LIN {X 0,Y 150.245,Z 335.769,A -85,B 0,C 180,E1 -24057.283,E2 -24057.283} C_VEL
LIN {X 0,Y 150.219,Z 335.772,A -85,B 0,C 180,E1 -24062.635,E2 -24062.635} C_VEL
LIN {X 0,Y 150.212,Z 335.771,A -85,B 0,C 180,E1 -24067.462,E2 -24067.462} C_VEL
LIN {X 0,Y 150.154,Z 335.78,A -85,B 0,C 180,E1 -24071.507,E2 -24071.507} C_VEL
LIN {X 0,Y 150.127,Z 335.783,A -85,B 0,C 180,E1 -24075.396,E2 -24075.396} C_VEL
LIN {X 0,Y 150.151,Z 335.779,A -85,B 0,C 180,E1 -24079.059,E2 -24079.059} C_VEL
LIN {X 0,Y 150.18,Z 335.776,A -85,B 0,C 180,E1 -24082.708,E2 -24082.708} C_VEL
LIN {X 0,Y 150.217,Z 335.772,A -85,B 0,C 180,E1 -24087.368,E2 -24087.368} C_VEL
LIN {X 0,Y 150.242,Z 335.765,A -85,B 0,C 180,E1 -24092.721,E2 -24092.721} C_VEL
LIN {X 0,Y 150.351,Z 335.756,A -85,B 0,C 180,E1 -24099.21,E2 -24099.21} C_VEL
LIN {X 0,Y 150.349,Z 335.756,A -85,B 0,C 180,E1 -24103.712,E2 -24103.712} C_VEL
LIN {X 0,Y 150.611,Z 335.72,A -85,B 0,C 180,E1 -24109.243,E2 -24109.243} C_VEL
LIN {X 0,Y 150.706,Z 335.711,A -85,B 0,C 180,E1 -24111.958,E2 -24111.958} C_VEL
LIN {X 0,Y 151.217,Z 335.647,A -85,B 0,C 180,E1 -24120,E2 -24120} C_VEL
LIN {X 0,Y 150.703,Z 335.711,A -85,B 0,C 180,E1 -24128.043,E2 -24128.043} C_VEL
LIN {X 0,Y 150.579,Z 335.726,A -85,B 0,C 180,E1 -24131.437,E2 -24131.437} C_VEL
LIN {X 0,Y 150.351,Z 335.755,A -85,B 0,C 180,E1 -24136.288,E2 -24136.288} C_VEL
LIN {X 0,Y 150.351,Z 335.753,A -85,B 0,C 180,E1 -24140.79,E2 -24140.79} C_VEL
LIN {X 0,Y 150.24,Z 335.748,A -85,B 0,C 180,E1 -24147.278,E2 -24147.278} C_VEL
LIN {X 0,Y 150.223,Z 335.774,A -85,B 0,C 180,E1 -24152.636,E2 -24152.636} C_VEL
LIN {X 0,Y 150.407,Z 335.951,A -85,B 0,C 180,E1 -24156.986,E2 -24156.986} C_VEL
LIN {X 0,Y 151.096,Z 339.515,A -85,B 0,C 180,E1 -24161.908,E2 -24161.908} C_VEL
LIN {X 0,Y 151.984,Z 343.974,A -85,B 0,C 180,E1 -24167.721,E2 -24167.721} C_VEL
LIN {X 0,Y 152.438,Z 347.108,A -85,B 0,C 180,E1 -24171.608,E2 -24171.608} C_VEL
LIN {X 0,Y 152.098,Z 348.347,A -85,B 0,C 180,E1 -24173.08,E2 -24173.08} C_VEL
LIN {X 0,Y 153.587,Z 362.688,A -85,B 0,C 180,E1 -24174.817,E2 -24174.817} C_VEL
LIN {X 0,Y 154.517,Z 375.98,A -85,B 0,C 180,E1 -24176.92,E2 -24176.92} C_VEL
LIN {X 0,Y 154.934,Z 388.273,A -85,B 0,C 180,E1 -24179.322,E2 -24179.322} C_VEL
LIN {X 0,Y 155.055,Z 399.237,A -85,B 0,C 180,E1 -24181.949,E2 -24181.949} C_VEL
LIN {X 0,Y 154.986,Z 410.057,A -85,B 0,C 180,E1 -24185.085,E2 -24185.085} C_VEL
LIN {X 0,Y 152.696,Z 419.643,A -85,B 0,C 180,E1 -24188.395,E2 -24188.395} C_VEL
LIN {X 0,Y 150.671,Z 428.608,A -85,B 0,C 180,E1 -24192.351,E2 -24192.351} C_VEL
LIN {X 0,Y 149.307,Z 435.832,A -85,B 0,C 180,E1 -24196.387,E2 -24196.387} C_VEL
LIN {X 0,Y 148.638,Z 441.612,A -85,B 0,C 180,E1 -24200.474,E2 -24200.474} C_VEL
LIN {X 0,Y 148.521,Z 446.113,A -85,B 0,C 180,E1 -24204.569,E2 -24204.569} C_VEL
LIN {X 0,Y 148.533,Z 448.434,A -85,B 0,C 180,E1 -24207.288,E2 -24207.288} C_VEL
LIN {X 0,Y 148.892,Z 450.302,A -85,B 0,C 180,E1 -24210,E2 -24210} C_VEL
LIN {X 0,Y 148.189,Z 452.535,A -85,B 0,C 180,E1 -24215.443,E2 -24215.443} C_VEL
LIN {X 0,Y 148.386,Z 453.179,A -85,B 0,C 180,E1 -24220.921,E2 -24220.921} C_VEL
LIN {X 0,Y 149.84,Z 452.386,A -85,B 0,C 180,E1 -24226.345,E2 -24226.345} C_VEL
LIN {X 0,Y 152.88,Z 450.2,A -85,B 0,C 180,E1 -24231.578,E2 -24231.578} C_VEL
LIN {X 0,Y 157.193,Z 446.504,A -85,B 0,C 180,E1 -24236.558,E2 -24236.558} C_VEL
LIN {X 0,Y 162.714,Z 441.245,A -85,B 0,C 180,E1 -24241.219,E2 -24241.219} C_VEL
LIN {X 0,Y 167.836,Z 436.146,A -85,B 0,C 180,E1 -24244.424,E2 -24244.424} C_VEL
LIN {X 0,Y 173.282,Z 429.984,A -85,B 0,C 180,E1 -24247.472,E2 -24247.472} C_VEL
LIN {X 0,Y 177.395,Z 423.553,A -85,B 0,C 180,E1 -24250.386,E2 -24250.386} C_VEL
LIN {X 0,Y 181.085,Z 416.172,A -85,B 0,C 180,E1 -24253.543,E2 -24253.543} C_VEL
LIN {X 0,Y 184.291,Z 407.788,A -85,B 0,C 180,E1 -24257.04,E2 -24257.04} C_VEL
LIN {X 0,Y 185.114,Z 404.915,A -85,B 0,C 180,E1 -24258.355,E2 -24258.355} C_VEL
LIN {X 0,Y 185.083,Z 402.347,A -85,B 0,C 180,E1 -24260.006,E2 -24260.006} C_VEL
LIN {X 0,Y 184.494,Z 400.473,A -85,B 0,C 180,E1 -24261.729,E2 -24261.729} C_VEL
LIN {X 0,Y 183.298,Z 399.467,A -85,B 0,C 180,E1 -24263.517,E2 -24263.517} C_VEL
LIN {X 0,Y 180.117,Z 398.092,A -85,B 0,C 180,E1 -24268.479,E2 -24268.479} C_VEL
LIN {X 0,Y 179.921,Z 397.396,A -85,B 0,C 180,E1 -24269.74,E2 -24269.74} C_VEL
LIN {X 0,Y 180.125,Z 395.776,A -85,B 0,C 180,E1 -24272.082,E2 -24272.082} C_VEL
LIN {X 0,Y 180.229,Z 394.714,A -85,B 0,C 180,E1 -24274.599,E2 -24274.599} C_VEL
LIN {X 0,Y 180.436,Z 394.168,A -85,B 0,C 180,E1 -24277.076,E2 -24277.076} C_VEL
LIN {X 0,Y 180.637,Z 394.859,A -85,B 0,C 180,E1 -24281.865,E2 -24281.865} C_VEL
LIN {X 0,Y 180.986,Z 395.569,A -85,B 0,C 180,E1 -24284.227,E2 -24284.227} C_VEL
LIN {X 0,Y 181.604,Z 398.314,A -85,B 0,C 180,E1 -24288.843,E2 -24288.843} C_VEL
LIN {X 0,Y 181.83,Z 401.361,A -85,B 0,C 180,E1 -24292.225,E2 -24292.225} C_VEL
LIN {X 0,Y 181.689,Z 403.801,A -85,B 0,C 180,E1 -24294.45,E2 -24294.45} C_VEL
LIN {X 0,Y 180.97,Z 407.418,A -85,B 0,C 180,E1 -24297.217,E2 -24297.217} C_VEL
LIN {X 0,Y 174.553,Z 414.57,A -85,B 0,C 180,E1 -24300,E2 -24300} C_VEL
LIN {X 0,Y 168.875,Z 420.089,A -85,B 0,C 180,E1 -24302.801,E2 -24302.801} C_VEL
LIN {X 0,Y 162.669,Z 425.365,A -85,B 0,C 180,E1 -24306.432,E2 -24306.432} C_VEL
LIN {X 0,Y 157.159,Z 429.256,A -85,B 0,C 180,E1 -24310.319,E2 -24310.319} C_VEL
LIN {X 0,Y 152.408,Z 431.935,A -85,B 0,C 180,E1 -24314.446,E2 -24314.446} C_VEL
LIN {X 0,Y 148.044,Z 433.624,A -85,B 0,C 180,E1 -24319.409,E2 -24319.409} C_VEL
LIN {X 0,Y 145.416,Z 433.971,A -85,B 0,C 180,E1 -24323.324,E2 -24323.324} C_VEL
LIN {X 0,Y 143.173,Z 433.396,A -85,B 0,C 180,E1 -24327.923,E2 -24327.923} C_VEL
LIN {X 0,Y 141.605,Z 431.564,A -85,B 0,C 180,E1 -24333.089,E2 -24333.089} C_VEL
LIN {X 0,Y 140.981,Z 428.174,A -85,B 0,C 180,E1 -24338.658,E2 -24338.658} C_VEL
LIN {X 0,Y 141.387,Z 423.269,A -85,B 0,C 180,E1 -24344.099,E2 -24344.099} C_VEL
LIN {X 0,Y 142.458,Z 417.277,A -85,B 0,C 180,E1 -24349.049,E2 -24349.049} C_VEL
LIN {X 0,Y 143.968,Z 410.137,A -85,B 0,C 180,E1 -24353.584,E2 -24353.584} C_VEL
LIN {X 0,Y 145.907,Z 402.46,A -85,B 0,C 180,E1 -24357.46,E2 -24357.46} C_VEL
LIN {X 0,Y 148.171,Z 393.253,A -85,B 0,C 180,E1 -24361.187,E2 -24361.187} C_VEL
LIN {X 0,Y 150.589,Z 383.793,A -85,B 0,C 180,E1 -24364.237,E2 -24364.237} C_VEL
LIN {X 0,Y 153.429,Z 371.561,A -85,B 0,C 180,E1 -24367.335,E2 -24367.335} C_VEL
LIN {X 0,Y 152.432,Z 365.897,A -85,B 0,C 180,E1 -24368.821,E2 -24368.821} C_VEL
LIN {X 0,Y 149.531,Z 354.899,A -85,B 0,C 180,E1 -24371.503,E2 -24371.503} C_VEL
LIN {X 0,Y 146.011,Z 344.016,A -85,B 0,C 180,E1 -24373.86,E2 -24373.86} C_VEL
LIN {X 0,Y 143.361,Z 336.628,A -85,B 0,C 180,E1 -24375.358,E2 -24375.358} C_VEL
LIN {X 0,Y 143.529,Z 336.608,A -85,B 0,C 180,E1 -24378.705,E2 -24378.705} C_VEL
LIN {X 0,Y 143.622,Z 336.6,A -85,B 0,C 180,E1 -24381.558,E2 -24381.558} C_VEL
LIN {X 0,Y 144.176,Z 336.519,A -85,B 0,C 180,E1 -24390,E2 -24390} C_VEL
LIN {X 0,Y 143.623,Z 336.592,A -85,B 0,C 180,E1 -24398.442,E2 -24398.442} C_VEL
LIN {X 0,Y 143.505,Z 336.609,A -85,B 0,C 180,E1 -24401.63,E2 -24401.63} C_VEL
LIN {X 0,Y 143.302,Z 336.634,A -85,B 0,C 180,E1 -24407.113,E2 -24407.113} C_VEL
LIN {X 0,Y 143.277,Z 336.633,A -85,B 0,C 180,E1 -24411.255,E2 -24411.255} C_VEL
LIN {X 0,Y 143.191,Z 336.649,A -85,B 0,C 180,E1 -24417.938,E2 -24417.938} C_VEL
LIN {X 0,Y 143.17,Z 336.65,A -85,B 0,C 180,E1 -24423.436,E2 -24423.436} C_VEL
LIN {X 0,Y 143.076,Z 336.658,A -85,B 0,C 180,E1 -24429.686,E2 -24429.686} C_VEL
LIN {X 0,Y 143.057,Z 336.665,A -85,B 0,C 180,E1 -24433.455,E2 -24433.455} C_VEL
LIN {X 0,Y 143.066,Z 336.658,A -85,B 0,C 180,E1 -24437.465,E2 -24437.465} C_VEL
LIN {X 0,Y 143.078,Z 336.662,A -85,B 0,C 180,E1 -24441.806,E2 -24441.806} C_VEL
LIN {X 0,Y 143.184,Z 336.648,A -85,B 0,C 180,E1 -24447.322,E2 -24447.322} C_VEL
LIN {X 0,Y 143.19,Z 336.644,A -85,B 0,C 180,E1 -24452.065,E2 -24452.065} C_VEL
LIN {X 0,Y 143.276,Z 336.637,A -85,B 0,C 180,E1 -24458.748,E2 -24458.748} C_VEL
LIN {X 0,Y 143.293,Z 336.632,A -85,B 0,C 180,E1 -24462.886,E2 -24462.886} C_VEL
LIN {X 0,Y 143.537,Z 336.602,A -85,B 0,C 180,E1 -24468.706,E2 -24468.706} C_VEL
LIN {X 0,Y 143.627,Z 336.593,A -85,B 0,C 180,E1 -24471.559,E2 -24471.559} C_VEL
LIN {X 0,Y 144.176,Z 336.524,A -85,B 0,C 180,E1 -24480,E2 -24480} C_VEL
LIN {X 0,Y 143.625,Z 336.593,A -85,B 0,C 180,E1 -24488.442,E2 -24488.442} C_VEL
LIN {X 0,Y 143.506,Z 336.607,A -85,B 0,C 180,E1 -24491.628,E2 -24491.628} C_VEL
LIN {X 0,Y 143.294,Z 336.635,A -85,B 0,C 180,E1 -24497.114,E2 -24497.114} C_VEL
LIN {X 0,Y 143.276,Z 336.633,A -85,B 0,C 180,E1 -24501.252,E2 -24501.252} C_VEL
LIN {X 0,Y 143.185,Z 336.629,A -85,B 0,C 180,E1 -24507.931,E2 -24507.931} C_VEL
LIN {X 0,Y 143.166,Z 336.653,A -85,B 0,C 180,E1 -24513.432,E2 -24513.432} C_VEL
LIN {X 0,Y 143.365,Z 336.834,A -85,B 0,C 180,E1 -24516.853,E2 -24516.853} C_VEL
LIN {X 0,Y 144.161,Z 341.144,A -85,B 0,C 180,E1 -24523.041,E2 -24523.041} C_VEL
LIN {X 0,Y 145.132,Z 345.655,A -85,B 0,C 180,E1 -24529.112,E2 -24529.112} C_VEL
LIN {X 0,Y 145.245,Z 347.987,A -85,B 0,C 180,E1 -24531.942,E2 -24531.942} C_VEL
LIN {X 0,Y 146.713,Z 360.951,A -85,B 0,C 180,E1 -24533.592,E2 -24533.592} C_VEL
LIN {X 0,Y 147.528,Z 374.304,A -85,B 0,C 180,E1 -24535.755,E2 -24535.755} C_VEL
LIN {X 0,Y 147.979,Z 385.945,A -85,B 0,C 180,E1 -24538.105,E2 -24538.105} C_VEL
LIN {X 0,Y 148.086,Z 397.385,A -85,B 0,C 180,E1 -24540.892,E2 -24540.892} C_VEL
LIN {X 0,Y 147.962,Z 408.129,A -85,B 0,C 180,E1 -24544.08,E2 -24544.08} C_VEL
LIN {X 0,Y 147.523,Z 411.986,A -85,B 0,C 180,E1 -24545.364,E2 -24545.364} C_VEL
LIN {X 0,Y 145.267,Z 420.792,A -85,B 0,C 180,E1 -24548.725,E2 -24548.725} C_VEL
LIN {X 0,Y 143.333,Z 429.463,A -85,B 0,C 180,E1 -24552.891,E2 -24552.891} C_VEL
LIN {X 0,Y 142.059,Z 436.408,A -85,B 0,C 180,E1 -24557.137,E2 -24557.137} C_VEL
LIN {X 0,Y 141.52,Z 441.927,A -85,B 0,C 180,E1 -24561.432,E2 -24561.432} C_VEL
LIN {X 0,Y 141.463,Z 446.196,A -85,B 0,C 180,E1 -24565.726,E2 -24565.726} C_VEL
LIN {X 0,Y 141.835,Z 449.329,A -85,B 0,C 180,E1 -24570,E2 -24570} C_VEL
LIN {X 0,Y 141.128,Z 451.694,A -85,B 0,C 180,E1 -24575.716,E2 -24575.716} C_VEL
LIN {X 0,Y 141.379,Z 452.562,A -85,B 0,C 180,E1 -24581.469,E2 -24581.469} C_VEL
LIN {X 0,Y 143.005,Z 451.956,A -85,B 0,C 180,E1 -24587.15,E2 -24587.15} C_VEL
LIN {X 0,Y 146.274,Z 449.958,A -85,B 0,C 180,E1 -24592.605,E2 -24592.605} C_VEL
LIN {X 0,Y 150.864,Z 446.527,A -85,B 0,C 180,E1 -24597.765,E2 -24597.765} C_VEL
LIN {X 0,Y 156.7,Z 441.521,A -85,B 0,C 180,E1 -24602.562,E2 -24602.562} C_VEL
LIN {X 0,Y 162.052,Z 436.665,A -85,B 0,C 180,E1 -24605.837,E2 -24605.837} C_VEL
LIN {X 0,Y 166.846,Z 431.825,A -85,B 0,C 180,E1 -24608.412,E2 -24608.412} C_VEL
LIN {X 0,Y 170.928,Z 426.317,A -85,B 0,C 180,E1 -24611.138,E2 -24611.138} C_VEL
LIN {X 0,Y 174.605,Z 420.247,A -85,B 0,C 180,E1 -24613.974,E2 -24613.974} C_VEL
LIN {X 0,Y 178.166,Z 412.97,A -85,B 0,C 180,E1 -24617.252,E2 -24617.252} C_VEL
LIN {X 0,Y 179.764,Z 408.96,A -85,B 0,C 180,E1 -24619.128,E2 -24619.128} C_VEL
LIN {X 0,Y 179.932,Z 405.737,A -85,B 0,C 180,E1 -24621.37,E2 -24621.37} C_VEL
LIN {X 0,Y 180.007,Z 401.346,A -85,B 0,C 180,E1 -24625.076,E2 -24625.076} C_VEL
LIN {X 0,Y 179.942,Z 399.637,A -85,B 0,C 180,E1 -24626.852,E2 -24626.852} C_VEL
LIN {X 0,Y 179.921,Z 397.396,A -85,B 0,C 180,E1 -24629.74,E2 -24629.74} C_VEL
LIN {X 0,Y 179.547,Z 396.738,A -85,B 0,C 180,E1 -24631.606,E2 -24631.606} C_VEL
LIN {X 0,Y 178.617,Z 397.022,A -85,B 0,C 180,E1 -24633.485,E2 -24633.485} C_VEL
LIN {X 0,Y 175.965,Z 399.453,A -85,B 0,C 180,E1 -24638.586,E2 -24638.586} C_VEL
LIN {X 0,Y 175.774,Z 399.815,A -85,B 0,C 180,E1 -24639.901,E2 -24639.901} C_VEL
LIN {X 0,Y 176.108,Z 400.68,A -85,B 0,C 180,E1 -24643.778,E2 -24643.778} C_VEL
LIN {X 0,Y 176.294,Z 401.749,A -85,B 0,C 180,E1 -24646.161,E2 -24646.161} C_VEL
LIN {X 0,Y 176.472,Z 403.124,A -85,B 0,C 180,E1 -24648.514,E2 -24648.514} C_VEL
LIN {X 0,Y 176.408,Z 405.939,A -85,B 0,C 180,E1 -24651.984,E2 -24651.984} C_VEL
LIN {X 0,Y 175.999,Z 408.249,A -85,B 0,C 180,E1 -24654.27,E2 -24654.27} C_VEL
LIN {X 0,Y 175.402,Z 410.284,A -85,B 0,C 180,E1 -24655.979,E2 -24655.979} C_VEL
LIN {X 0,Y 167.712,Z 417.965,A -85,B 0,C 180,E1 -24659.253,E2 -24659.253} C_VEL
LIN {X 0,Y 161.208,Z 423.488,A -85,B 0,C 180,E1 -24662.498,E2 -24662.498} C_VEL
LIN {X 0,Y 155.456,Z 427.697,A -85,B 0,C 180,E1 -24665.953,E2 -24665.953} C_VEL
LIN {X 0,Y 149.863,Z 431.104,A -85,B 0,C 180,E1 -24669.992,E2 -24669.992} C_VEL
LIN {X 0,Y 145.055,Z 433.318,A -85,B 0,C 180,E1 -24674.299,E2 -24674.299} C_VEL
LIN {X 0,Y 141.099,Z 434.435,A -85,B 0,C 180,E1 -24678.848,E2 -24678.848} C_VEL
LIN {X 0,Y 137.749,Z 434.434,A -85,B 0,C 180,E1 -24684.089,E2 -24684.089} C_VEL
LIN {X 0,Y 135.809,Z 433.538,A -85,B 0,C 180,E1 -24688.389,E2 -24688.389} C_VEL
LIN {X 0,Y 134.464,Z 431.572,A -85,B 0,C 180,E1 -24693.251,E2 -24693.251} C_VEL
LIN {X 0,Y 133.878,Z 427.9,A -85,B 0,C 180,E1 -24699.046,E2 -24699.046} C_VEL
LIN {X 0,Y 134.418,Z 422.569,A -85,B 0,C 180,E1 -24704.897,E2 -24704.897} C_VEL
LIN {X 0,Y 135.591,Z 416.362,A -85,B 0,C 180,E1 -24709.941,E2 -24709.941} C_VEL
LIN {X 0,Y 137.354,Z 408.436,A -85,B 0,C 180,E1 -24714.951,E2 -24714.951} C_VEL
LIN {X 0,Y 139.457,Z 400.349,A -85,B 0,C 180,E1 -24718.95,E2 -24718.95} C_VEL
LIN {X 0,Y 142.096,Z 390.282,A -85,B 0,C 180,E1 -24722.907,E2 -24722.907} C_VEL
LIN {X 0,Y 144.743,Z 379.879,A -85,B 0,C 180,E1 -24726.136,E2 -24726.136} C_VEL
LIN {X 0,Y 146.341,Z 373.192,A -85,B 0,C 180,E1 -24727.835,E2 -24727.835} C_VEL
LIN {X 0,Y 146.462,Z 371.459,A -85,B 0,C 180,E1 -24728.281,E2 -24728.281} C_VEL
LIN {X 0,Y 144.025,Z 360.858,A -85,B 0,C 180,E1 -24731.138,E2 -24731.138} C_VEL
LIN {X 0,Y 140.443,Z 348.913,A -85,B 0,C 180,E1 -24734.024,E2 -24734.024} C_VEL
LIN {X 0,Y 136.353,Z 337.528,A -85,B 0,C 180,E1 -24736.531,E2 -24736.531} C_VEL
LIN {X 0,Y 136.547,Z 337.483,A -85,B 0,C 180,E1 -24741.117,E2 -24741.117} C_VEL
LIN {X 0,Y 137.133,Z 337.396,A -85,B 0,C 180,E1 -24750,E2 -24750} C_VEL
LIN {X 0,Y 136.55,Z 337.475,A -85,B 0,C 180,E1 -24758.882,E2 -24758.882} C_VEL
LIN {X 0,Y 136.441,Z 337.489,A -85,B 0,C 180,E1 -24761.89,E2 -24761.89} C_VEL
LIN {X 0,Y 136.243,Z 337.514,A -85,B 0,C 180,E1 -24768.03,E2 -24768.03} C_VEL
LIN {X 0,Y 136.199,Z 337.515,A -85,B 0,C 180,E1 -24771.749,E2 -24771.749} C_VEL
LIN {X 0,Y 136.101,Z 337.529,A -85,B 0,C 180,E1 -24778.617,E2 -24778.617} C_VEL
LIN {X 0,Y 136.079,Z 337.534,A -85,B 0,C 180,E1 -24784.619,E2 -24784.619} C_VEL
LIN {X 0,Y 136.051,Z 337.532,A -85,B 0,C 180,E1 -24789.208,E2 -24789.208} C_VEL
LIN {X 0,Y 135.999,Z 337.545,A -85,B 0,C 180,E1 -24793.658,E2 -24793.658} C_VEL
LIN {X 0,Y 136.005,Z 337.539,A -85,B 0,C 180,E1 -24797.797,E2 -24797.797} C_VEL
LIN {X 0,Y 136.028,Z 337.541,A -85,B 0,C 180,E1 -24801.685,E2 -24801.685} C_VEL
LIN {X 0,Y 136.056,Z 337.533,A -85,B 0,C 180,E1 -24805.74,E2 -24805.74} C_VEL
LIN {X 0,Y 136.145,Z 337.521,A -85,B 0,C 180,E1 -24812.317,E2 -24812.317} C_VEL
LIN {X 0,Y 136.243,Z 337.513,A -85,B 0,C 180,E1 -24818.833,E2 -24818.833} C_VEL
LIN {X 0,Y 136.246,Z 337.514,A -85,B 0,C 180,E1 -24825.054,E2 -24825.054} C_VEL
LIN {X 0,Y 136.427,Z 337.487,A -85,B 0,C 180,E1 -24828.178,E2 -24828.178} C_VEL
LIN {X 0,Y 136.552,Z 337.473,A -85,B 0,C 180,E1 -24831.118,E2 -24831.118} C_VEL
LIN {X 0,Y 137.133,Z 337.401,A -85,B 0,C 180,E1 -24840,E2 -24840} C_VEL
LIN {X 0,Y 136.551,Z 337.476,A -85,B 0,C 180,E1 -24848.883,E2 -24848.883} C_VEL
LIN {X 0,Y 136.442,Z 337.487,A -85,B 0,C 180,E1 -24851.891,E2 -24851.891} C_VEL
LIN {X 0,Y 136.238,Z 337.514,A -85,B 0,C 180,E1 -24858.031,E2 -24858.031} C_VEL
LIN {X 0,Y 136.197,Z 337.515,A -85,B 0,C 180,E1 -24861.746,E2 -24861.746} C_VEL
LIN {X 0,Y 136.094,Z 337.515,A -85,B 0,C 180,E1 -24868.61,E2 -24868.61} C_VEL
LIN {X 0,Y 136.322,Z 337.618,A -85,B 0,C 180,E1 -24876.591,E2 -24876.591} C_VEL
LIN {X 0,Y 136.947,Z 341.085,A -85,B 0,C 180,E1 -24881.848,E2 -24881.848} C_VEL
LIN {X 0,Y 137.946,Z 345.763,A -85,B 0,C 180,E1 -24888.523,E2 -24888.523} C_VEL
LIN {X 0,Y 138.196,Z 347.298,A -85,B 0,C 180,E1 -24890.634,E2 -24890.634} C_VEL
LIN {X 0,Y 139.643,Z 357.54,A -85,B 0,C 180,E1 -24892.052,E2 -24892.052} C_VEL
LIN {X 0,Y 140.584,Z 370.636,A -85,B 0,C 180,E1 -24894.158,E2 -24894.158} C_VEL
LIN {X 0,Y 141.026,Z 381.698,A -85,B 0,C 180,E1 -24896.351,E2 -24896.351} C_VEL
LIN {X 0,Y 141.176,Z 393.28,A -85,B 0,C 180,E1 -24899.14,E2 -24899.14} C_VEL
LIN {X 0,Y 141.021,Z 404.853,A -85,B 0,C 180,E1 -24902.549,E2 -24902.549} C_VEL
LIN {X 0,Y 140.782,Z 410.704,A -85,B 0,C 180,E1 -24904.544,E2 -24904.544} C_VEL
LIN {X 0,Y 138.239,Z 420.331,A -85,B 0,C 180,E1 -24908.371,E2 -24908.371} C_VEL
LIN {X 0,Y 136.262,Z 428.973,A -85,B 0,C 180,E1 -24912.748,E2 -24912.748} C_VEL
LIN {X 0,Y 134.996,Z 435.881,A -85,B 0,C 180,E1 -24917.217,E2 -24917.217} C_VEL
LIN {X 0,Y 134.465,Z 442.154,A -85,B 0,C 180,E1 -24922.493,E2 -24922.493} C_VEL
LIN {X 0,Y 134.455,Z 446.187,A -85,B 0,C 180,E1 -24927.004,E2 -24927.004} C_VEL
LIN {X 0,Y 134.78,Z 448.284,A -85,B 0,C 180,E1 -24930,E2 -24930} C_VEL
LIN {X 0,Y 134.122,Z 450.673,A -85,B 0,C 180,E1 -24935.369,E2 -24935.369} C_VEL
LIN {X 0,Y 134.097,Z 451.549,A -85,B 0,C 180,E1 -24939.046,E2 -24939.046} C_VEL
LIN {X 0,Y 135.12,Z 451.865,A -85,B 0,C 180,E1 -24945.074,E2 -24945.074} C_VEL
LIN {X 0,Y 137.813,Z 450.799,A -85,B 0,C 180,E1 -24950.915,E2 -24950.915} C_VEL
LIN {X 0,Y 142.041,Z 448.286,A -85,B 0,C 180,E1 -24956.443,E2 -24956.443} C_VEL
LIN {X 0,Y 147.522,Z 444.355,A -85,B 0,C 180,E1 -24961.604,E2 -24961.604} C_VEL
LIN {X 0,Y 152.538,Z 440.353,A -85,B 0,C 180,E1 -24965.165,E2 -24965.165} C_VEL
LIN {X 0,Y 158.383,Z 435.381,A -85,B 0,C 180,E1 -24968.406,E2 -24968.406} C_VEL
LIN {X 0,Y 162.259,Z 431.556,A -85,B 0,C 180,E1 -24970.52,E2 -24970.52} C_VEL
LIN {X 0,Y 166.675,Z 425.883,A -85,B 0,C 180,E1 -24973.488,E2 -24973.488} C_VEL
LIN {X 0,Y 170.991,Z 419.074,A -85,B 0,C 180,E1 -24976.85,E2 -24976.85} C_VEL
LIN {X 0,Y 174.308,Z 412.689,A -85,B 0,C 180,E1 -24980.003,E2 -24980.003} C_VEL
LIN {X 0,Y 174.842,Z 408.305,A -85,B 0,C 180,E1 -24983.507,E2 -24983.507} C_VEL
LIN {X 0,Y 174.992,Z 405.928,A -85,B 0,C 180,E1 -24985.787,E2 -24985.787} C_VEL
LIN {X 0,Y 175.135,Z 402.528,A -85,B 0,C 180,E1 -24990.17,E2 -24990.17} C_VEL
LIN {X 0,Y 175.375,Z 401.39,A -85,B 0,C 180,E1 -24991.841,E2 -24991.841} C_VEL
LIN {X 0,Y 175.572,Z 400.417,A -85,B 0,C 180,E1 -24993.875,E2 -24993.875} C_VEL
LIN {X 0,Y 175.793,Z 399.63,A -85,B 0,C 180,E1 -24996.856,E2 -24996.856} C_VEL
LIN {X 0,Y 175.774,Z 399.815,A -85,B 0,C 180,E1 -24999.901,E2 -24999.901} C_VEL
LIN {X 0,Y 175.394,Z 400.701,A -85,B 0,C 180,E1 -25001.803,E2 -25001.803} C_VEL
LIN {X 0,Y 174.352,Z 402.414,A -85,B 0,C 180,E1 -25003.643,E2 -25003.643} C_VEL
LIN {X 0,Y 171.237,Z 407.858,A -85,B 0,C 180,E1 -25008.563,E2 -25008.563} C_VEL
LIN {X 0,Y 170.97,Z 408.845,A -85,B 0,C 180,E1 -25009.863,E2 -25009.863} C_VEL
LIN {X 0,Y 170.559,Z 411.305,A -85,B 0,C 180,E1 -25012.899,E2 -25012.899} C_VEL
LIN {X 0,Y 170.12,Z 412.478,A -85,B 0,C 180,E1 -25014.073,E2 -25014.073} C_VEL
LIN {X 0,Y 169.36,Z 413.599,A -85,B 0,C 180,E1 -25014.839,E2 -25014.839} C_VEL
LIN {X 0,Y 161.74,Z 420.404,A -85,B 0,C 180,E1 -25018.04,E2 -25018.04} C_VEL
LIN {X 0,Y 154.674,Z 425.775,A -85,B 0,C 180,E1 -25021.547,E2 -25021.547} C_VEL
LIN {X 0,Y 148.23,Z 429.87,A -85,B 0,C 180,E1 -25025.441,E2 -25025.441} C_VEL
LIN {X 0,Y 142.563,Z 432.736,A -85,B 0,C 180,E1 -25029.613,E2 -25029.613} C_VEL
LIN {X 0,Y 136.998,Z 434.685,A -85,B 0,C 180,E1 -25034.862,E2 -25034.862} C_VEL
LIN {X 0,Y 133.7,Z 435.214,A -85,B 0,C 180,E1 -25038.882,E2 -25038.882} C_VEL
LIN {X 0,Y 130.63,Z 434.873,A -85,B 0,C 180,E1 -25043.848,E2 -25043.848} C_VEL
LIN {X 0,Y 128.24,Z 433.274,A -85,B 0,C 180,E1 -25049.553,E2 -25049.553} C_VEL
LIN {X 0,Y 126.993,Z 430.189,A -85,B 0,C 180,E1 -25055.672,E2 -25055.672} C_VEL
LIN {X 0,Y 126.91,Z 425.77,A -85,B 0,C 180,E1 -25061.646,E2 -25061.646} C_VEL
LIN {X 0,Y 127.755,Z 419.993,A -85,B 0,C 180,E1 -25067.318,E2 -25067.318} C_VEL
LIN {X 0,Y 128.951,Z 414.346,A -85,B 0,C 180,E1 -25071.669,E2 -25071.669} C_VEL
LIN {X 0,Y 131.038,Z 405.803,A -85,B 0,C 180,E1 -25076.86,E2 -25076.86} C_VEL
LIN {X 0,Y 133.206,Z 397.599,A -85,B 0,C 180,E1 -25080.788,E2 -25080.788} C_VEL
LIN {X 0,Y 136.129,Z 386.982,A -85,B 0,C 180,E1 -25084.79,E2 -25084.79} C_VEL
LIN {X 0,Y 139.023,Z 375.735,A -85,B 0,C 180,E1 -25088.11,E2 -25088.11} C_VEL
LIN {X 0,Y 139.524,Z 372.436,A -85,B 0,C 180,E1 -25088.967,E2 -25088.967} C_VEL
LIN {X 0,Y 137.02,Z 361.66,A -85,B 0,C 180,E1 -25092.076,E2 -25092.076} C_VEL
LIN {X 0,Y 133.465,Z 349.866,A -85,B 0,C 180,E1 -25095.145,E2 -25095.145} C_VEL
LIN {X 0,Y 129.463,Z 338.909,A -85,B 0,C 180,E1 -25097.726,E2 -25097.726} C_VEL
LIN {X 0,Y 129.369,Z 338.373,A -85,B 0,C 180,E1 -25097.917,E2 -25097.917} C_VEL
LIN {X 0,Y 129.47,Z 338.363,A -85,B 0,C 180,E1 -25100.628,E2 -25100.628} C_VEL
LIN {X 0,Y 130.088,Z 338.273,A -85,B 0,C 180,E1 -25110,E2 -25110} C_VEL
LIN {X 0,Y 129.473,Z 338.356,A -85,B 0,C 180,E1 -25119.372,E2 -25119.372} C_VEL
LIN {X 0,Y 129.344,Z 338.372,A -85,B 0,C 180,E1 -25122.553,E2 -25122.553} C_VEL
LIN {X 0,Y 129.154,Z 338.396,A -85,B 0,C 180,E1 -25129.056,E2 -25129.056} C_VEL
LIN {X 0,Y 129.109,Z 338.397,A -85,B 0,C 180,E1 -25132.398,E2 -25132.398} C_VEL
LIN {X 0,Y 129.036,Z 338.408,A -85,B 0,C 180,E1 -25139.374,E2 -25139.374} C_VEL
LIN {X 0,Y 128.993,Z 338.416,A -85,B 0,C 180,E1 -25145.19,E2 -25145.19} C_VEL
LIN {X 0,Y 128.951,Z 338.42,A -85,B 0,C 180,E1 -25150.845,E2 -25150.845} C_VEL
LIN {X 0,Y 128.922,Z 338.424,A -85,B 0,C 180,E1 -25155.128,E2 -25155.128} C_VEL
LIN {X 0,Y 128.943,Z 338.423,A -85,B 0,C 180,E1 -25159.736,E2 -25159.736} C_VEL
LIN {X 0,Y 128.96,Z 338.415,A -85,B 0,C 180,E1 -25164.832,E2 -25164.832} C_VEL
LIN {X 0,Y 129.017,Z 338.413,A -85,B 0,C 180,E1 -25170.643,E2 -25170.643} C_VEL
LIN {X 0,Y 129.028,Z 338.409,A -85,B 0,C 180,E1 -25174.167,E2 -25174.167} C_VEL
LIN {X 0,Y 129.108,Z 338.402,A -85,B 0,C 180,E1 -25177.729,E2 -25177.729} C_VEL
LIN {X 0,Y 129.149,Z 338.392,A -85,B 0,C 180,E1 -25180.944,E2 -25180.944} C_VEL
LIN {X 0,Y 129.35,Z 338.369,A -85,B 0,C 180,E1 -25187.962,E2 -25187.962} C_VEL
LIN {X 0,Y 129.474,Z 338.353,A -85,B 0,C 180,E1 -25190.628,E2 -25190.628} C_VEL
LIN {X 0,Y 130.088,Z 338.279,A -85,B 0,C 180,E1 -25200,E2 -25200} C_VEL
LIN {X 0,Y 129.474,Z 338.357,A -85,B 0,C 180,E1 -25209.372,E2 -25209.372} C_VEL
LIN {X 0,Y 129.345,Z 338.37,A -85,B 0,C 180,E1 -25212.553,E2 -25212.553} C_VEL
LIN {X 0,Y 129.15,Z 338.396,A -85,B 0,C 180,E1 -25219.057,E2 -25219.057} C_VEL
LIN {X 0,Y 129.109,Z 338.393,A -85,B 0,C 180,E1 -25222.399,E2 -25222.399} C_VEL
LIN {X 0,Y 129.018,Z 338.401,A -85,B 0,C 180,E1 -25229.358,E2 -25229.358} C_VEL
LIN {X 0,Y 129.26,Z 338.501,A -85,B 0,C 180,E1 -25236.512,E2 -25236.512} C_VEL
LIN {X 0,Y 129.963,Z 342.288,A -85,B 0,C 180,E1 -25242.527,E2 -25242.527} C_VEL
LIN {X 0,Y 130.933,Z 346.6,A -85,B 0,C 180,E1 -25248.988,E2 -25248.988} C_VEL
LIN {X 0,Y 130.954,Z 346.811,A -85,B 0,C 180,E1 -25249.227,E2 -25249.227} C_VEL
LIN {X 0,Y 132.554,Z 353.665,A -85,B 0,C 180,E1 -25250.31,E2 -25250.31} C_VEL
LIN {X 0,Y 133.597,Z 366.413,A -85,B 0,C 180,E1 -25252.354,E2 -25252.354} C_VEL
LIN {X 0,Y 134.128,Z 380.26,A -85,B 0,C 180,E1 -25255.155,E2 -25255.155} C_VEL
LIN {X 0,Y 134.213,Z 391.447,A -85,B 0,C 180,E1 -25257.928,E2 -25257.928} C_VEL
LIN {X 0,Y 134.018,Z 402.963,A -85,B 0,C 180,E1 -25261.411,E2 -25261.411} C_VEL
LIN {X 0,Y 133.82,Z 410.05,A -85,B 0,C 180,E1 -25263.925,E2 -25263.925} C_VEL
LIN {X 0,Y 131.671,Z 418.151,A -85,B 0,C 180,E1 -25267.234,E2 -25267.234} C_VEL
LIN {X 0,Y 129.483,Z 427.047,A -85,B 0,C 180,E1 -25271.814,E2 -25271.814} C_VEL
LIN {X 0,Y 128.095,Z 434.223,A -85,B 0,C 180,E1 -25276.516,E2 -25276.516} C_VEL
LIN {X 0,Y 127.509,Z 439.074,A -85,B 0,C 180,E1 -25280.482,E2 -25280.482} C_VEL
LIN {X 0,Y 127.423,Z 443.727,A -85,B 0,C 180,E1 -25285.254,E2 -25285.254} C_VEL
LIN {X 0,Y 127.727,Z 447.194,A -85,B 0,C 180,E1 -25290,E2 -25290} C_VEL
LIN {X 0,Y 127.09,Z 449.685,A -85,B 0,C 180,E1 -25295.501,E2 -25295.501} C_VEL
LIN {X 0,Y 127.067,Z 450.769,A -85,B 0,C 180,E1 -25299.551,E2 -25299.551} C_VEL
LIN {X 0,Y 128.263,Z 451.265,A -85,B 0,C 180,E1 -25305.901,E2 -25305.901} C_VEL
LIN {X 0,Y 131.188,Z 450.4,A -85,B 0,C 180,E1 -25312.025,E2 -25312.025} C_VEL
LIN {X 0,Y 135.68,Z 448.166,A -85,B 0,C 180,E1 -25317.787,E2 -25317.787} C_VEL
LIN {X 0,Y 141.511,Z 444.442,A -85,B 0,C 180,E1 -25323.114,E2 -25323.114} C_VEL
LIN {X 0,Y 146.809,Z 440.693,A -85,B 0,C 180,E1 -25326.756,E2 -25326.756} C_VEL
LIN {X 0,Y 155.016,Z 434.187,A -85,B 0,C 180,E1 -25331.102,E2 -25331.102} C_VEL
LIN {X 0,Y 159.595,Z 429.313,A -85,B 0,C 180,E1 -25333.914,E2 -25333.914} C_VEL
LIN {X 0,Y 164.613,Z 422.835,A -85,B 0,C 180,E1 -25337.432,E2 -25337.432} C_VEL
LIN {X 0,Y 168.221,Z 417.117,A -85,B 0,C 180,E1 -25340.433,E2 -25340.433} C_VEL
LIN {X 0,Y 168.896,Z 415.672,A -85,B 0,C 180,E1 -25341.378,E2 -25341.378} C_VEL
LIN {X 0,Y 169.519,Z 412.195,A -85,B 0,C 180,E1 -25344.52,E2 -25344.52} C_VEL
LIN {X 0,Y 169.9,Z 409.553,A -85,B 0,C 180,E1 -25347.469,E2 -25347.469} C_VEL
LIN {X 0,Y 170.515,Z 405.984,A -85,B 0,C 180,E1 -25353.039,E2 -25353.039} C_VEL
LIN {X 0,Y 170.739,Z 405.044,A -85,B 0,C 180,E1 -25355.693,E2 -25355.693} C_VEL
LIN {X 0,Y 170.857,Z 404.775,A -85,B 0,C 180,E1 -25358.271,E2 -25358.271} C_VEL
LIN {X 0,Y 171.015,Z 405.55,A -85,B 0,C 180,E1 -25363.281,E2 -25363.281} C_VEL
LIN {X 0,Y 171.061,Z 406.44,A -85,B 0,C 180,E1 -25365.729,E2 -25365.729} C_VEL
LIN {X 0,Y 171.135,Z 407.696,A -85,B 0,C 180,E1 -25368.151,E2 -25368.151} C_VEL
LIN {X 0,Y 170.97,Z 408.845,A -85,B 0,C 180,E1 -25369.863,E2 -25369.863} C_VEL
LIN {X 0,Y 170.417,Z 409.969,A -85,B 0,C 180,E1 -25370.867,E2 -25370.867} C_VEL
LIN {X 0,Y 168.478,Z 412.255,A -85,B 0,C 180,E1 -25372.055,E2 -25372.055} C_VEL
LIN {X 0,Y 163.485,Z 416.775,A -85,B 0,C 180,E1 -25373.751,E2 -25373.751} C_VEL
LIN {X 0,Y 159.984,Z 419.601,A -85,B 0,C 180,E1 -25374.972,E2 -25374.972} C_VEL
LIN {X 0,Y 151.698,Z 425.682,A -85,B 0,C 180,E1 -25378.672,E2 -25378.672} C_VEL
LIN {X 0,Y 144.199,Z 430.216,A -85,B 0,C 180,E1 -25382.793,E2 -25382.793} C_VEL
LIN {X 0,Y 139.683,Z 432.476,A -85,B 0,C 180,E1 -25385.775,E2 -25385.775} C_VEL
LIN {X 0,Y 135.264,Z 434.212,A -85,B 0,C 180,E1 -25389.174,E2 -25389.174} C_VEL
LIN {X 0,Y 130.319,Z 435.525,A -85,B 0,C 180,E1 -25393.895,E2 -25393.895} C_VEL
LIN {X 0,Y 125.808,Z 435.787,A -85,B 0,C 180,E1 -25399.583,E2 -25399.583} C_VEL
LIN {X 0,Y 123.216,Z 435.061,A -85,B 0,C 180,E1 -25404.13,E2 -25404.13} C_VEL
LIN {X 0,Y 121.109,Z 433.322,A -85,B 0,C 180,E1 -25409.488,E2 -25409.488} C_VEL
LIN {X 0,Y 119.869,Z 430.002,A -85,B 0,C 180,E1 -25415.895,E2 -25415.895} C_VEL
LIN {X 0,Y 119.866,Z 425.056,A -85,B 0,C 180,E1 -25422.395,E2 -25422.395} C_VEL
LIN {X 0,Y 120.805,Z 419.293,A -85,B 0,C 180,E1 -25428.067,E2 -25428.067} C_VEL
LIN {X 0,Y 122.381,Z 412.128,A -85,B 0,C 180,E1 -25433.511,E2 -25433.511} C_VEL
LIN {X 0,Y 124.826,Z 403.093,A -85,B 0,C 180,E1 -25438.826,E2 -25438.826} C_VEL
LIN {X 0,Y 127.411,Z 393.625,A -85,B 0,C 180,E1 -25443.176,E2 -25443.176} C_VEL
LIN {X 0,Y 130.312,Z 383.378,A -85,B 0,C 180,E1 -25446.844,E2 -25446.844} C_VEL
LIN {X 0,Y 132.668,Z 374.294,A -85,B 0,C 180,E1 -25449.454,E2 -25449.454} C_VEL
LIN {X 0,Y 130.837,Z 365.442,A -85,B 0,C 180,E1 -25452.207,E2 -25452.207} C_VEL
LIN {X 0,Y 127.371,Z 353.38,A -85,B 0,C 180,E1 -25455.623,E2 -25455.623} C_VEL
LIN {X 0,Y 122.964,Z 341.423,A -85,B 0,C 180,E1 -25458.773,E2 -25458.773} C_VEL
LIN {X 0,Y 122.352,Z 339.247,A -85,B 0,C 180,E1 -25459.284,E2 -25459.284} C_VEL
LIN {X 0,Y 122.595,Z 339.217,A -85,B 0,C 180,E1 -25466.714,E2 -25466.714} C_VEL
LIN {X 0,Y 123.041,Z 339.15,A -85,B 0,C 180,E1 -25470,E2 -25470} C_VEL
LIN {X 0,Y 122.422,Z 339.234,A -85,B 0,C 180,E1 -25476.593,E2 -25476.593} C_VEL
LIN {X 0,Y 122.409,Z 339.237,A -85,B 0,C 180,E1 -25479.918,E2 -25479.918} C_VEL
LIN {X 0,Y 122.24,Z 339.255,A -85,B 0,C 180,E1 -25483.296,E2 -25483.296} C_VEL
LIN {X 0,Y 122.046,Z 339.281,A -85,B 0,C 180,E1 -25490.213,E2 -25490.213} C_VEL
LIN {X 0,Y 121.984,Z 339.286,A -85,B 0,C 180,E1 -25493.785,E2 -25493.785} C_VEL
LIN {X 0,Y 121.942,Z 339.29,A -85,B 0,C 180,E1 -25500.174,E2 -25500.174} C_VEL
LIN {X 0,Y 121.913,Z 339.297,A -85,B 0,C 180,E1 -25506.19,E2 -25506.19} C_VEL
LIN {X 0,Y 121.885,Z 339.301,A -85,B 0,C 180,E1 -25511.445,E2 -25511.445} C_VEL
LIN {X 0,Y 121.873,Z 339.302,A -85,B 0,C 180,E1 -25518.562,E2 -25518.562} C_VEL
LIN {X 0,Y 121.912,Z 339.293,A -85,B 0,C 180,E1 -25524.797,E2 -25524.797} C_VEL
LIN {X 0,Y 121.927,Z 339.297,A -85,B 0,C 180,E1 -25529.839,E2 -25529.839} C_VEL
LIN {X 0,Y 121.983,Z 339.289,A -85,B 0,C 180,E1 -25536.216,E2 -25536.216} C_VEL
LIN {X 0,Y 122.043,Z 339.279,A -85,B 0,C 180,E1 -25539.787,E2 -25539.787} C_VEL
LIN {X 0,Y 122.098,Z 339.274,A -85,B 0,C 180,E1 -25543.274,E2 -25543.274} C_VEL
LIN {X 0,Y 122.401,Z 339.233,A -85,B 0,C 180,E1 -25550.082,E2 -25550.082} C_VEL
LIN {X 0,Y 122.599,Z 339.209,A -85,B 0,C 180,E1 -25556.714,E2 -25556.714} C_VEL
LIN {X 0,Y 123.041,Z 339.157,A -85,B 0,C 180,E1 -25560,E2 -25560} C_VEL
LIN {X 0,Y 122.419,Z 339.23,A -85,B 0,C 180,E1 -25566.594,E2 -25566.594} C_VEL
LIN {X 0,Y 122.324,Z 339.245,A -85,B 0,C 180,E1 -25572.386,E2 -25572.386} C_VEL
LIN {X 0,Y 122.105,Z 339.275,A -85,B 0,C 180,E1 -25576.726,E2 -25576.726} C_VEL
LIN {X 0,Y 122.028,Z 339.273,A -85,B 0,C 180,E1 -25582.854,E2 -25582.854} C_VEL
LIN {X 0,Y 121.936,Z 339.287,A -85,B 0,C 180,E1 -25590.167,E2 -25590.167} C_VEL
LIN {X 0,Y 122.222,Z 339.332,A -85,B 0,C 180,E1 -25596.386,E2 -25596.386} C_VEL
LIN {X 0,Y 122.982,Z 343.481,A -85,B 0,C 180,E1 -25603.296,E2 -25603.296} C_VEL
LIN {X 0,Y 123.632,Z 346.293,A -85,B 0,C 180,E1 -25607.647,E2 -25607.647} C_VEL
LIN {X 0,Y 124.595,Z 349.556,A -85,B 0,C 180,E1 -25608.214,E2 -25608.214} C_VEL
LIN {X 0,Y 126.087,Z 355.337,A -85,B 0,C 180,E1 -25609.263,E2 -25609.263} C_VEL
LIN {X 0,Y 126.931,Z 367.414,A -85,B 0,C 180,E1 -25611.379,E2 -25611.379} C_VEL
LIN {X 0,Y 127.294,Z 380.275,A -85,B 0,C 180,E1 -25614.167,E2 -25614.167} C_VEL
LIN {X 0,Y 127.304,Z 392.466,A -85,B 0,C 180,E1 -25617.434,E2 -25617.434} C_VEL
LIN {X 0,Y 127.024,Z 402.995,A -85,B 0,C 180,E1 -25620.854,E2 -25620.854} C_VEL
LIN {X 0,Y 126.686,Z 410.363,A -85,B 0,C 180,E1 -25623.653,E2 -25623.653} C_VEL
LIN {X 0,Y 124.232,Z 419.134,A -85,B 0,C 180,E1 -25627.551,E2 -25627.551} C_VEL
LIN {X 0,Y 122.154,Z 427.771,A -85,B 0,C 180,E1 -25632.419,E2 -25632.419} C_VEL
LIN {X 0,Y 120.848,Z 434.692,A -85,B 0,C 180,E1 -25637.403,E2 -25637.403} C_VEL
LIN {X 0,Y 120.386,Z 440.64,A -85,B 0,C 180,E1 -25642.954,E2 -25642.954} C_VEL
LIN {X 0,Y 120.505,Z 444.965,A -85,B 0,C 180,E1 -25648.329,E2 -25648.329} C_VEL
LIN {X 0,Y 120.677,Z 446.073,A -85,B 0,C 180,E1 -25650,E2 -25650} C_VEL
LIN {X 0,Y 120.063,Z 448.678,A -85,B 0,C 180,E1 -25655.664,E2 -25655.664} C_VEL
LIN {X 0,Y 120.059,Z 449.919,A -85,B 0,C 180,E1 -25660.114,E2 -25660.114} C_VEL
LIN {X 0,Y 121.421,Z 450.658,A -85,B 0,C 180,E1 -25666.823,E2 -25666.823} C_VEL
LIN {X 0,Y 124.621,Z 449.992,A -85,B 0,C 180,E1 -25673.252,E2 -25673.252} C_VEL
LIN {X 0,Y 129.407,Z 447.96,A -85,B 0,C 180,E1 -25679.261,E2 -25679.261} C_VEL
LIN {X 0,Y 135.597,Z 444.566,A -85,B 0,C 180,E1 -25684.76,E2 -25684.76} C_VEL
LIN {X 0,Y 141.194,Z 441.003,A -85,B 0,C 180,E1 -25688.477,E2 -25688.477} C_VEL
LIN {X 0,Y 147.565,Z 436.511,A -85,B 0,C 180,E1 -25691.819,E2 -25691.819} C_VEL
LIN {X 0,Y 151.746,Z 433.063,A -85,B 0,C 180,E1 -25694.005,E2 -25694.005} C_VEL
LIN {X 0,Y 157.424,Z 427.017,A -85,B 0,C 180,E1 -25697.658,E2 -25697.658} C_VEL
LIN {X 0,Y 162.269,Z 420.769,A -85,B 0,C 180,E1 -25701.224,E2 -25701.224} C_VEL
LIN {X 0,Y 163.047,Z 419.572,A -85,B 0,C 180,E1 -25701.986,E2 -25701.986} C_VEL
LIN {X 0,Y 163.858,Z 416.822,A -85,B 0,C 180,E1 -25704.58,E2 -25704.58} C_VEL
LIN {X 0,Y 164.213,Z 415.357,A -85,B 0,C 180,E1 -25706.194,E2 -25706.194} C_VEL
LIN {X 0,Y 164.634,Z 413.184,A -85,B 0,C 180,E1 -25709.185,E2 -25709.185} C_VEL
LIN {X 0,Y 165.304,Z 410.829,A -85,B 0,C 180,E1 -25713.232,E2 -25713.232} C_VEL
LIN {X 0,Y 165.496,Z 410.192,A -85,B 0,C 180,E1 -25714.87,E2 -25714.87} C_VEL
LIN {X 0,Y 165.656,Z 409.686,A -85,B 0,C 180,E1 -25718.965,E2 -25718.965} C_VEL
LIN {X 0,Y 165.689,Z 410.174,A -85,B 0,C 180,E1 -25722.727,E2 -25722.727} C_VEL
LIN {X 0,Y 165.648,Z 410.903,A -85,B 0,C 180,E1 -25725.252,E2 -25725.252} C_VEL
LIN {X 0,Y 165.613,Z 412.016,A -85,B 0,C 180,E1 -25727.749,E2 -25727.749} C_VEL
LIN {X 0,Y 165.28,Z 413.457,A -85,B 0,C 180,E1 -25730.207,E2 -25730.207} C_VEL
LIN {X 0,Y 164.624,Z 415.328,A -85,B 0,C 180,E1 -25732.641,E2 -25732.641} C_VEL
LIN {X 0,Y 164.186,Z 416.036,A -85,B 0,C 180,E1 -25733.33,E2 -25733.33} C_VEL
LIN {X 0,Y 159.984,Z 419.601,A -85,B 0,C 180,E1 -25734.972,E2 -25734.972} C_VEL
LIN {X 0,Y 156.135,Z 422.407,A -85,B 0,C 180,E1 -25736.258,E2 -25736.258} C_VEL
LIN {X 0,Y 148.621,Z 426.782,A -85,B 0,C 180,E1 -25738.06,E2 -25738.06} C_VEL
LIN {X 0,Y 141.114,Z 430.449,A -85,B 0,C 180,E1 -25740.138,E2 -25740.138} C_VEL
LIN {X 0,Y 137.372,Z 432.11,A -85,B 0,C 180,E1 -25741.867,E2 -25741.867} C_VEL
LIN {X 0,Y 131.076,Z 434.597,A -85,B 0,C 180,E1 -25746.156,E2 -25746.156} C_VEL
LIN {X 0,Y 126.981,Z 435.768,A -85,B 0,C 180,E1 -25749.557,E2 -25749.557} C_VEL
LIN {X 0,Y 122.934,Z 436.391,A -85,B 0,C 180,E1 -25753.619,E2 -25753.619} C_VEL
LIN {X 0,Y 118.859,Z 436.248,A -85,B 0,C 180,E1 -25758.902,E2 -25758.902} C_VEL
LIN {X 0,Y 115.466,Z 434.874,A -85,B 0,C 180,E1 -25765.218,E2 -25765.218} C_VEL
LIN {X 0,Y 113.356,Z 432.097,A -85,B 0,C 180,E1 -25771.951,E2 -25771.951} C_VEL
LIN {X 0,Y 112.602,Z 427.977,A -85,B 0,C 180,E1 -25778.619,E2 -25778.619} C_VEL
LIN {X 0,Y 113.101,Z 422.506,A -85,B 0,C 180,E1 -25785.141,E2 -25785.141} C_VEL
LIN {X 0,Y 114.476,Z 415.795,A -85,B 0,C 180,E1 -25791.158,E2 -25791.158} C_VEL
LIN {X 0,Y 116.186,Z 408.876,A -85,B 0,C 180,E1 -25796.049,E2 -25796.049} C_VEL
LIN {X 0,Y 118.551,Z 400.606,A -85,B 0,C 180,E1 -25800.72,E2 -25800.72} C_VEL
LIN {X 0,Y 121.437,Z 390.61,A -85,B 0,C 180,E1 -25805.191,E2 -25805.191} C_VEL
LIN {X 0,Y 124.469,Z 379.873,A -85,B 0,C 180,E1 -25808.902,E2 -25808.902} C_VEL
LIN {X 0,Y 125.753,Z 374.703,A -85,B 0,C 180,E1 -25810.408,E2 -25810.408} C_VEL
LIN {X 0,Y 123.615,Z 365.409,A -85,B 0,C 180,E1 -25813.485,E2 -25813.485} C_VEL
LIN {X 0,Y 120.762,Z 355.428,A -85,B 0,C 180,E1 -25816.539,E2 -25816.539} C_VEL
LIN {X 0,Y 116.492,Z 343.375,A -85,B 0,C 180,E1 -25820.011,E2 -25820.011} C_VEL
LIN {X 0,Y 115.35,Z 340.124,A -85,B 0,C 180,E1 -25820.907,E2 -25820.907} C_VEL
LIN {X 0,Y 115.993,Z 340.028,A -85,B 0,C 180,E1 -25830,E2 -25830} C_VEL
LIN {X 0,Y 115.363,Z 340.112,A -85,B 0,C 180,E1 -25836.998,E2 -25836.998} C_VEL
LIN {X 0,Y 115.249,Z 340.127,A -85,B 0,C 180,E1 -25842.66,E2 -25842.66} C_VEL
LIN {X 0,Y 115.012,Z 340.158,A -85,B 0,C 180,E1 -25847.79,E2 -25847.79} C_VEL
LIN {X 0,Y 114.947,Z 340.162,A -85,B 0,C 180,E1 -25853.493,E2 -25853.493} C_VEL
LIN {X 0,Y 114.869,Z 340.171,A -85,B 0,C 180,E1 -25861.069,E2 -25861.069} C_VEL
LIN {X 0,Y 114.803,Z 340.18,A -85,B 0,C 180,E1 -25867.748,E2 -25867.748} C_VEL
LIN {X 0,Y 114.795,Z 340.185,A -85,B 0,C 180,E1 -25872.722,E2 -25872.722} C_VEL
LIN {X 0,Y 114.795,Z 340.18,A -85,B 0,C 180,E1 -25877.667,E2 -25877.667} C_VEL
LIN {X 0,Y 114.789,Z 340.185,A -85,B 0,C 180,E1 -25882.744,E2 -25882.744} C_VEL
LIN {X 0,Y 114.857,Z 340.178,A -85,B 0,C 180,E1 -25888.943,E2 -25888.943} C_VEL
LIN {X 0,Y 114.948,Z 340.166,A -85,B 0,C 180,E1 -25896.508,E2 -25896.508} C_VEL
LIN {X 0,Y 115.005,Z 340.155,A -85,B 0,C 180,E1 -25902.209,E2 -25902.209} C_VEL
LIN {X 0,Y 115.313,Z 340.115,A -85,B 0,C 180,E1 -25909.465,E2 -25909.465} C_VEL
LIN {X 0,Y 115.523,Z 340.091,A -85,B 0,C 180,E1 -25916.513,E2 -25916.513} C_VEL
LIN {X 0,Y 115.992,Z 340.035,A -85,B 0,C 180,E1 -25920,E2 -25920} C_VEL
LIN {X 0,Y 115.361,Z 340.111,A -85,B 0,C 180,E1 -25926.999,E2 -25926.999} C_VEL
LIN {X 0,Y 115.257,Z 340.123,A -85,B 0,C 180,E1 -25932.673,E2 -25932.673} C_VEL
LIN {X 0,Y 115.009,Z 340.158,A -85,B 0,C 180,E1 -25937.791,E2 -25937.791} C_VEL
LIN {X 0,Y 114.946,Z 340.151,A -85,B 0,C 180,E1 -25943.489,E2 -25943.489} C_VEL
LIN {X 0,Y 114.878,Z 340.171,A -85,B 0,C 180,E1 -25951.074,E2 -25951.074} C_VEL
LIN {X 0,Y 115.183,Z 340.285,A -85,B 0,C 180,E1 -25956.506,E2 -25956.506} C_VEL
LIN {X 0,Y 115.911,Z 344.155,A -85,B 0,C 180,E1 -25963.315,E2 -25963.315} C_VEL
LIN {X 0,Y 116.26,Z 345.614,A -85,B 0,C 180,E1 -25965.803,E2 -25965.803} C_VEL
LIN {X 0,Y 117.374,Z 349.206,A -85,B 0,C 180,E1 -25966.551,E2 -25966.551} C_VEL
LIN {X 0,Y 119.587,Z 356.882,A -85,B 0,C 180,E1 -25968.163,E2 -25968.163} C_VEL
LIN {X 0,Y 120.282,Z 369.27,A -85,B 0,C 180,E1 -25970.549,E2 -25970.549} C_VEL
LIN {X 0,Y 120.488,Z 380.919,A -85,B 0,C 180,E1 -25973.282,E2 -25973.282} C_VEL
LIN {X 0,Y 120.364,Z 393.142,A -85,B 0,C 180,E1 -25976.811,E2 -25976.811} C_VEL
LIN {X 0,Y 119.988,Z 403.881,A -85,B 0,C 180,E1 -25980.565,E2 -25980.565} C_VEL
LIN {X 0,Y 119.719,Z 409.709,A -85,B 0,C 180,E1 -25982.938,E2 -25982.938} C_VEL
LIN {X 0,Y 117.26,Z 418.488,A -85,B 0,C 180,E1 -25987.072,E2 -25987.072} C_VEL
LIN {X 0,Y 115.106,Z 427.101,A -85,B 0,C 180,E1 -25992.225,E2 -25992.225} C_VEL
LIN {X 0,Y 113.789,Z 434.017,A -85,B 0,C 180,E1 -25997.516,E2 -25997.516} C_VEL
LIN {X 0,Y 113.364,Z 439.508,A -85,B 0,C 180,E1 -26002.878,E2 -26002.878} C_VEL
LIN {X 0,Y 113.471,Z 443.731,A -85,B 0,C 180,E1 -26008.225,E2 -26008.225} C_VEL
LIN {X 0,Y 113.647,Z 444.876,A -85,B 0,C 180,E1 -26010,E2 -26010} C_VEL
LIN {X 0,Y 113.045,Z 447.625,A -85,B 0,C 180,E1 -26015.887,E2 -26015.887} C_VEL
LIN {X 0,Y 113.077,Z 449.039,A -85,B 0,C 180,E1 -26020.746,E2 -26020.746} C_VEL
LIN {X 0,Y 114.622,Z 449.966,A -85,B 0,C 180,E1 -26027.853,E2 -26027.853} C_VEL
LIN {X 0,Y 118.104,Z 449.564,A -85,B 0,C 180,E1 -26034.617,E2 -26034.617} C_VEL
LIN {X 0,Y 123.231,Z 447.774,A -85,B 0,C 180,E1 -26040.883,E2 -26040.883} C_VEL
LIN {X 0,Y 129.821,Z 444.601,A -85,B 0,C 180,E1 -26046.548,E2 -26046.548} C_VEL
LIN {X 0,Y 137.874,Z 439.996,A -85,B 0,C 180,E1 -26051.504,E2 -26051.504} C_VEL
LIN {X 0,Y 144.628,Z 435.47,A -85,B 0,C 180,E1 -26054.798,E2 -26054.798} C_VEL
LIN {X 0,Y 148.659,Z 432.044,A -85,B 0,C 180,E1 -26057.12,E2 -26057.12} C_VEL
LIN {X 0,Y 154.297,Z 426.316,A -85,B 0,C 180,E1 -26060.744,E2 -26060.744} C_VEL
LIN {X 0,Y 156.054,Z 424.298,A -85,B 0,C 180,E1 -26062.011,E2 -26062.011} C_VEL
LIN {X 0,Y 157.536,Z 422.304,A -85,B 0,C 180,E1 -26063.42,E2 -26063.42} C_VEL
LIN {X 0,Y 158.437,Z 419.713,A -85,B 0,C 180,E1 -26066.326,E2 -26066.326} C_VEL
LIN {X 0,Y 159.287,Z 416.689,A -85,B 0,C 180,E1 -26070.965,E2 -26070.965} C_VEL
LIN {X 0,Y 159.946,Z 415.178,A -85,B 0,C 180,E1 -26073.934,E2 -26073.934} C_VEL
LIN {X 0,Y 160.183,Z 414.411,A -85,B 0,C 180,E1 -26077.128,E2 -26077.128} C_VEL
LIN {X 0,Y 160.217,Z 414.302,A -85,B 0,C 180,E1 -26079.456,E2 -26079.456} C_VEL
LIN {X 0,Y 160.139,Z 414.561,A -85,B 0,C 180,E1 -26082.109,E2 -26082.109} C_VEL
LIN {X 0,Y 160.052,Z 415.234,A -85,B 0,C 180,E1 -26085.026,E2 -26085.026} C_VEL
LIN {X 0,Y 159.921,Z 416.064,A -85,B 0,C 180,E1 -26087.306,E2 -26087.306} C_VEL
LIN {X 0,Y 159.424,Z 417.396,A -85,B 0,C 180,E1 -26089.843,E2 -26089.843} C_VEL
LIN {X 0,Y 158.994,Z 418.239,A -85,B 0,C 180,E1 -26091.1,E2 -26091.1} C_VEL
LIN {X 0,Y 157.517,Z 419.677,A -85,B 0,C 180,E1 -26092.307,E2 -26092.307} C_VEL
LIN {X 0,Y 149.701,Z 425.28,A -85,B 0,C 180,E1 -26095.462,E2 -26095.462} C_VEL
LIN {X 0,Y 143.128,Z 429.217,A -85,B 0,C 180,E1 -26098.585,E2 -26098.585} C_VEL
LIN {X 0,Y 137.372,Z 432.11,A -85,B 0,C 180,E1 -26101.867,E2 -26101.867} C_VEL
LIN {X 0,Y 133.704,Z 433.561,A -85,B 0,C 180,E1 -26103.738,E2 -26103.738} C_VEL
LIN {X 0,Y 126.488,Z 435.588,A -85,B 0,C 180,E1 -26106.608,E2 -26106.608} C_VEL
LIN {X 0,Y 119.557,Z 436.834,A -85,B 0,C 180,E1 -26109.85,E2 -26109.85} C_VEL
LIN {X 0,Y 116.452,Z 437.047,A -85,B 0,C 180,E1 -26112.28,E2 -26112.28} C_VEL
LIN {X 0,Y 111.433,Z 436.528,A -85,B 0,C 180,E1 -26118.906,E2 -26118.906} C_VEL
LIN {X 0,Y 108.397,Z 434.975,A -85,B 0,C 180,E1 -26124.809,E2 -26124.809} C_VEL
LIN {X 0,Y 106.22,Z 431.884,A -85,B 0,C 180,E1 -26131.959,E2 -26131.959} C_VEL
LIN {X 0,Y 105.526,Z 427.347,A -85,B 0,C 180,E1 -26139.247,E2 -26139.247} C_VEL
LIN {X 0,Y 105.937,Z 422.863,A -85,B 0,C 180,E1 -26144.708,E2 -26144.708} C_VEL
LIN {X 0,Y 107.025,Z 417.319,A -85,B 0,C 180,E1 -26150.12,E2 -26150.12} C_VEL
LIN {X 0,Y 108.959,Z 409.608,A -85,B 0,C 180,E1 -26156.067,E2 -26156.067} C_VEL
LIN {X 0,Y 111.741,Z 400.142,A -85,B 0,C 180,E1 -26161.706,E2 -26161.706} C_VEL
LIN {X 0,Y 114.442,Z 391.112,A -85,B 0,C 180,E1 -26165.914,E2 -26165.914} C_VEL
LIN {X 0,Y 117.283,Z 381.592,A -85,B 0,C 180,E1 -26169.426,E2 -26169.426} C_VEL
LIN {X 0,Y 118.825,Z 376.031,A -85,B 0,C 180,E1 -26171.143,E2 -26171.143} C_VEL
LIN {X 0,Y 116.815,Z 366.776,A -85,B 0,C 180,E1 -26174.445,E2 -26174.445} C_VEL
LIN {X 0,Y 114.169,Z 357.444,A -85,B 0,C 180,E1 -26177.558,E2 -26177.558} C_VEL
LIN {X 0,Y 110.528,Z 346.836,A -85,B 0,C 180,E1 -26180.853,E2 -26180.853} C_VEL
LIN {X 0,Y 108.301,Z 340.995,A -85,B 0,C 180,E1 -26182.66,E2 -26182.66} C_VEL
LIN {X 0,Y 108.918,Z 340.909,A -85,B 0,C 180,E1 -26190,E2 -26190} C_VEL
LIN {X 0,Y 108.303,Z 340.99,A -85,B 0,C 180,E1 -26197.457,E2 -26197.457} C_VEL
LIN {X 0,Y 108.171,Z 341.008,A -85,B 0,C 180,E1 -26202.951,E2 -26202.951} C_VEL
LIN {X 0,Y 107.904,Z 341.043,A -85,B 0,C 180,E1 -26209.006,E2 -26209.006} C_VEL
LIN {X 0,Y 107.858,Z 341.047,A -85,B 0,C 180,E1 -26214.185,E2 -26214.185} C_VEL
LIN {X 0,Y 107.795,Z 341.054,A -85,B 0,C 180,E1 -26222.052,E2 -26222.052} C_VEL
LIN {X 0,Y 107.707,Z 341.062,A -85,B 0,C 180,E1 -26228.464,E2 -26228.464} C_VEL
LIN {X 0,Y 107.679,Z 341.066,A -85,B 0,C 180,E1 -26235.886,E2 -26235.886} C_VEL
LIN {X 0,Y 107.689,Z 341.071,A -85,B 0,C 180,E1 -26241.55,E2 -26241.55} C_VEL
LIN {X 0,Y 107.793,Z 341.057,A -85,B 0,C 180,E1 -26248.561,E2 -26248.561} C_VEL
LIN {X 0,Y 107.912,Z 341.043,A -85,B 0,C 180,E1 -26256.998,E2 -26256.998} C_VEL
LIN {X 0,Y 108.016,Z 341.03,A -85,B 0,C 180,E1 -26264.915,E2 -26264.915} C_VEL
LIN {X 0,Y 108.23,Z 340.998,A -85,B 0,C 180,E1 -26268.767,E2 -26268.767} C_VEL
LIN {X 0,Y 108.447,Z 340.973,A -85,B 0,C 180,E1 -26276.285,E2 -26276.285} C_VEL
LIN {X 0,Y 108.917,Z 340.916,A -85,B 0,C 180,E1 -26280,E2 -26280} C_VEL
LIN {X 0,Y 108.301,Z 340.992,A -85,B 0,C 180,E1 -26287.458,E2 -26287.458} C_VEL
LIN {X 0,Y 108.177,Z 341.004,A -85,B 0,C 180,E1 -26292.961,E2 -26292.961} C_VEL
LIN {X 0,Y 107.903,Z 341.043,A -85,B 0,C 180,E1 -26299.006,E2 -26299.006} C_VEL
LIN {X 0,Y 107.855,Z 341.029,A -85,B 0,C 180,E1 -26304.179,E2 -26304.179} C_VEL
LIN {X 0,Y 107.827,Z 341.053,A -85,B 0,C 180,E1 -26312.078,E2 -26312.078} C_VEL
LIN {X 0,Y 108.125,Z 341.041,A -85,B 0,C 180,E1 -26316.337,E2 -26316.337} C_VEL
LIN {X 0,Y 108.897,Z 345.017,A -85,B 0,C 180,E1 -26323.771,E2 -26323.771} C_VEL
LIN {X 0,Y 110.062,Z 348.689,A -85,B 0,C 180,E1 -26324.621,E2 -26324.621} C_VEL
LIN {X 0,Y 113.03,Z 358.016,A -85,B 0,C 180,E1 -26326.846,E2 -26326.846} C_VEL
LIN {X 0,Y 113.62,Z 370.147,A -85,B 0,C 180,E1 -26329.417,E2 -26329.417} C_VEL
LIN {X 0,Y 113.678,Z 382.893,A -85,B 0,C 180,E1 -26332.729,E2 -26332.729} C_VEL
LIN {X 0,Y 113.398,Z 395.162,A -85,B 0,C 180,E1 -26336.63,E2 -26336.63} C_VEL
LIN {X 0,Y 112.905,Z 405.447,A -85,B 0,C 180,E1 -26340.629,E2 -26340.629} C_VEL
LIN {X 0,Y 112.781,Z 408.882,A -85,B 0,C 180,E1 -26342.136,E2 -26342.136} C_VEL
LIN {X 0,Y 110.775,Z 416.115,A -85,B 0,C 180,E1 -26345.645,E2 -26345.645} C_VEL
LIN {X 0,Y 108.367,Z 425.055,A -85,B 0,C 180,E1 -26351.079,E2 -26351.079} C_VEL
LIN {X 0,Y 106.907,Z 432.246,A -85,B 0,C 180,E1 -26356.698,E2 -26356.698} C_VEL
LIN {X 0,Y 106.354,Z 437.99,A -85,B 0,C 180,E1 -26362.405,E2 -26362.405} C_VEL
LIN {X 0,Y 106.44,Z 442.43,A -85,B 0,C 180,E1 -26368.108,E2 -26368.108} C_VEL
LIN {X 0,Y 106.617,Z 443.641,A -85,B 0,C 180,E1 -26370,E2 -26370} C_VEL
LIN {X 0,Y 106.038,Z 446.512,A -85,B 0,C 180,E1 -26376.183,E2 -26376.183} C_VEL
LIN {X 0,Y 106.122,Z 448.131,A -85,B 0,C 180,E1 -26381.46,E2 -26381.46} C_VEL
LIN {X 0,Y 107.873,Z 449.266,A -85,B 0,C 180,E1 -26389.011,E2 -26389.011} C_VEL
LIN {X 0,Y 111.667,Z 449.064,A -85,B 0,C 180,E1 -26396.14,E2 -26396.14} C_VEL
LIN {X 0,Y 117.17,Z 447.536,A -85,B 0,C 180,E1 -26402.673,E2 -26402.673} C_VEL
LIN {X 0,Y 124.179,Z 444.659,A -85,B 0,C 180,E1 -26408.503,E2 -26408.503} C_VEL
LIN {X 0,Y 132.645,Z 440.32,A -85,B 0,C 180,E1 -26413.534,E2 -26413.534} C_VEL
LIN {X 0,Y 139.661,Z 436.051,A -85,B 0,C 180,E1 -26416.859,E2 -26416.859} C_VEL
LIN {X 0,Y 143.866,Z 432.818,A -85,B 0,C 180,E1 -26419.218,E2 -26419.218} C_VEL
LIN {X 0,Y 148.436,Z 428.779,A -85,B 0,C 180,E1 -26422.01,E2 -26422.01} C_VEL
LIN {X 0,Y 151.486,Z 425.582,A -85,B 0,C 180,E1 -26424.282,E2 -26424.282} C_VEL
LIN {X 0,Y 152.412,Z 423.817,A -85,B 0,C 180,E1 -26426.403,E2 -26426.403} C_VEL
LIN {X 0,Y 153.151,Z 421.687,A -85,B 0,C 180,E1 -26429.683,E2 -26429.683} C_VEL
LIN {X 0,Y 153.924,Z 420.04,A -85,B 0,C 180,E1 -26432.832,E2 -26432.832} C_VEL
LIN {X 0,Y 154.38,Z 418.993,A -85,B 0,C 180,E1 -26435.813,E2 -26435.813} C_VEL
LIN {X 0,Y 154.527,Z 418.61,A -85,B 0,C 180,E1 -26438.663,E2 -26438.663} C_VEL
LIN {X 0,Y 154.317,Z 418.946,A -85,B 0,C 180,E1 -26443.019,E2 -26443.019} C_VEL
LIN {X 0,Y 154.032,Z 419.871,A -85,B 0,C 180,E1 -26446.812,E2 -26446.812} C_VEL
LIN {X 0,Y 153.438,Z 421.055,A -85,B 0,C 180,E1 -26449.443,E2 -26449.443} C_VEL
LIN {X 0,Y 152.19,Z 422.203,A -85,B 0,C 180,E1 -26450.698,E2 -26450.698} C_VEL
LIN {X 0,Y 142.972,Z 427.981,A -85,B 0,C 180,E1 -26454.358,E2 -26454.358} C_VEL
LIN {X 0,Y 137.25,Z 430.99,A -85,B 0,C 180,E1 -26457.064,E2 -26457.064} C_VEL
LIN {X 0,Y 131.845,Z 433.374,A -85,B 0,C 180,E1 -26460.061,E2 -26460.061} C_VEL
LIN {X 0,Y 126.723,Z 435.178,A -85,B 0,C 180,E1 -26463.357,E2 -26463.357} C_VEL
LIN {X 0,Y 120.685,Z 436.634,A -85,B 0,C 180,E1 -26468.114,E2 -26468.114} C_VEL
LIN {X 0,Y 116.452,Z 437.047,A -85,B 0,C 180,E1 -26472.28,E2 -26472.28} C_VEL
LIN {X 0,Y 113.551,Z 437.098,A -85,B 0,C 180,E1 -26474.846,E2 -26474.846} C_VEL
LIN {X 0,Y 107.651,Z 436.59,A -85,B 0,C 180,E1 -26478.972,E2 -26478.972} C_VEL
LIN {X 0,Y 103.24,Z 435.64,A -85,B 0,C 180,E1 -26482.531,E2 -26482.531} C_VEL
LIN {X 0,Y 100.922,Z 434.552,A -85,B 0,C 180,E1 -26485.525,E2 -26485.525} C_VEL
LIN {X 0,Y 100.46,Z 434.075,A -85,B 0,C 180,E1 -26486.587,E2 -26486.587} C_VEL
LIN {X 0,Y 99.128,Z 431.743,A -85,B 0,C 180,E1 -26491.703,E2 -26491.703} C_VEL
LIN {X 0,Y 98.43,Z 427.811,A -85,B 0,C 180,E1 -26498.241,E2 -26498.241} C_VEL
LIN {X 0,Y 98.9,Z 422.236,A -85,B 0,C 180,E1 -26505.285,E2 -26505.285} C_VEL
LIN {X 0,Y 100.367,Z 415.402,A -85,B 0,C 180,E1 -26511.972,E2 -26511.972} C_VEL
LIN {X 0,Y 102.315,Z 408.222,A -85,B 0,C 180,E1 -26517.512,E2 -26517.512} C_VEL
LIN {X 0,Y 105.149,Z 398.911,A -85,B 0,C 180,E1 -26523.141,E2 -26523.141} C_VEL
LIN {X 0,Y 108.601,Z 388.104,A -85,B 0,C 180,E1 -26528.155,E2 -26528.155} C_VEL
LIN {X 0,Y 111.909,Z 376.659,A -85,B 0,C 180,E1 -26532.213,E2 -26532.213} C_VEL
LIN {X 0,Y 109.869,Z 367.681,A -85,B 0,C 180,E1 -26535.648,E2 -26535.648} C_VEL
LIN {X 0,Y 107.49,Z 359.098,A -85,B 0,C 180,E1 -26538.736,E2 -26538.736} C_VEL
LIN {X 0,Y 103.53,Z 347.598,A -85,B 0,C 180,E1 -26542.687,E2 -26542.687} C_VEL
LIN {X 0,Y 101.359,Z 342.194,A -85,B 0,C 180,E1 -26544.529,E2 -26544.529} C_VEL
LIN {X 0,Y 101.331,Z 341.861,A -85,B 0,C 180,E1 -26544.777,E2 -26544.777} C_VEL
LIN {X 0,Y 101.846,Z 341.789,A -85,B 0,C 180,E1 -26550,E2 -26550} C_VEL
LIN {X 0,Y 101.241,Z 341.87,A -85,B 0,C 180,E1 -26557.981,E2 -26557.981} C_VEL
LIN {X 0,Y 101.1,Z 341.888,A -85,B 0,C 180,E1 -26563.294,E2 -26563.294} C_VEL
LIN {X 0,Y 100.816,Z 341.924,A -85,B 0,C 180,E1 -26570.399,E2 -26570.399} C_VEL
LIN {X 0,Y 100.774,Z 341.931,A -85,B 0,C 180,E1 -26574.959,E2 -26574.959} C_VEL
LIN {X 0,Y 100.7,Z 341.94,A -85,B 0,C 180,E1 -26583.124,E2 -26583.124} C_VEL
LIN {X 0,Y 100.654,Z 341.942,A -85,B 0,C 180,E1 -26589.821,E2 -26589.821} C_VEL
LIN {X 0,Y 100.651,Z 341.942,A -85,B 0,C 180,E1 -26595.713,E2 -26595.713} C_VEL
LIN {X 0,Y 100.628,Z 341.95,A -85,B 0,C 180,E1 -26601.056,E2 -26601.056} C_VEL
LIN {X 0,Y 100.689,Z 341.94,A -85,B 0,C 180,E1 -26606.887,E2 -26606.887} C_VEL
LIN {X 0,Y 100.787,Z 341.928,A -85,B 0,C 180,E1 -26615.268,E2 -26615.268} C_VEL
LIN {X 0,Y 100.814,Z 341.923,A -85,B 0,C 180,E1 -26619.601,E2 -26619.601} C_VEL
LIN {X 0,Y 101.129,Z 341.884,A -85,B 0,C 180,E1 -26627.967,E2 -26627.967} C_VEL
LIN {X 0,Y 101.237,Z 341.873,A -85,B 0,C 180,E1 -26632.02,E2 -26632.02} C_VEL
LIN {X 0,Y 101.845,Z 341.797,A -85,B 0,C 180,E1 -26640.001,E2 -26640.001} C_VEL
LIN {X 0,Y 101.241,Z 341.872,A -85,B 0,C 180,E1 -26647.981,E2 -26647.981} C_VEL
LIN {X 0,Y 101.105,Z 341.884,A -85,B 0,C 180,E1 -26653.302,E2 -26653.302} C_VEL
LIN {X 0,Y 100.815,Z 341.923,A -85,B 0,C 180,E1 -26660.4,E2 -26660.4} C_VEL
LIN {X 0,Y 100.776,Z 341.904,A -85,B 0,C 180,E1 -26664.959,E2 -26664.959} C_VEL
LIN {X 0,Y 100.853,Z 341.925,A -85,B 0,C 180,E1 -26673.883,E2 -26673.883} C_VEL
LIN {X 0,Y 101.123,Z 342.115,A -85,B 0,C 180,E1 -26676.83,E2 -26676.83} C_VEL
LIN {X 0,Y 101.572,Z 344.571,A -85,B 0,C 180,E1 -26681.589,E2 -26681.589} C_VEL
LIN {X 0,Y 102.708,Z 348.109,A -85,B 0,C 180,E1 -26682.454,E2 -26682.454} C_VEL
LIN {X 0,Y 106.441,Z 359.476,A -85,B 0,C 180,E1 -26685.493,E2 -26685.493} C_VEL
LIN {X 0,Y 106.958,Z 367.925,A -85,B 0,C 180,E1 -26687.444,E2 -26687.444} C_VEL
LIN {X 0,Y 106.926,Z 379.585,A -85,B 0,C 180,E1 -26690.496,E2 -26690.496} C_VEL
LIN {X 0,Y 106.626,Z 391.052,A -85,B 0,C 180,E1 -26694.199,E2 -26694.199} C_VEL
LIN {X 0,Y 106.093,Z 402.038,A -85,B 0,C 180,E1 -26698.494,E2 -26698.494} C_VEL
LIN {X 0,Y 105.489,Z 410.021,A -85,B 0,C 180,E1 -26702.201,E2 -26702.201} C_VEL
LIN {X 0,Y 102.866,Z 418.537,A -85,B 0,C 180,E1 -26706.868,E2 -26706.868} C_VEL
LIN {X 0,Y 100.756,Z 426.938,A -85,B 0,C 180,E1 -26712.756,E2 -26712.756} C_VEL
LIN {X 0,Y 99.683,Z 432.586,A -85,B 0,C 180,E1 -26717.789,E2 -26717.789} C_VEL
LIN {X 0,Y 99.335,Z 437.834,A -85,B 0,C 180,E1 -26723.57,E2 -26723.57} C_VEL
LIN {X 0,Y 99.608,Z 442.345,A -85,B 0,C 180,E1 -26730,E2 -26730} C_VEL
LIN {X 0,Y 99.044,Z 445.394,A -85,B 0,C 180,E1 -26736.574,E2 -26736.574} C_VEL
LIN {X 0,Y 99.195,Z 447.142,A -85,B 0,C 180,E1 -26742.272,E2 -26742.272} C_VEL
LIN {X 0,Y 101.18,Z 448.512,A -85,B 0,C 180,E1 -26750.323,E2 -26750.323} C_VEL
LIN {X 0,Y 105.31,Z 448.563,A -85,B 0,C 180,E1 -26757.85,E2 -26757.85} C_VEL
LIN {X 0,Y 111.712,Z 447.11,A -85,B 0,C 180,E1 -26765.129,E2 -26765.129} C_VEL
LIN {X 0,Y 118.693,Z 444.644,A -85,B 0,C 180,E1 -26770.642,E2 -26770.642} C_VEL
LIN {X 0,Y 127.602,Z 440.642,A -85,B 0,C 180,E1 -26775.726,E2 -26775.726} C_VEL
LIN {X 0,Y 134.882,Z 436.645,A -85,B 0,C 180,E1 -26779.072,E2 -26779.072} C_VEL
LIN {X 0,Y 139.261,Z 433.617,A -85,B 0,C 180,E1 -26781.466,E2 -26781.466} C_VEL
LIN {X 0,Y 143.662,Z 430.118,A -85,B 0,C 180,E1 -26784.052,E2 -26784.052} C_VEL
LIN {X 0,Y 145.379,Z 428.57,A -85,B 0,C 180,E1 -26785.268,E2 -26785.268} C_VEL
LIN {X 0,Y 146.302,Z 427.323,A -85,B 0,C 180,E1 -26786.819,E2 -26786.819} C_VEL
LIN {X 0,Y 147.031,Z 425.761,A -85,B 0,C 180,E1 -26789.361,E2 -26789.361} C_VEL
LIN {X 0,Y 148.19,Z 423.497,A -85,B 0,C 180,E1 -26794.303,E2 -26794.303} C_VEL
LIN {X 0,Y 148.554,Z 422.711,A -85,B 0,C 180,E1 -26797.76,E2 -26797.76} C_VEL
LIN {X 0,Y 148.494,Z 422.607,A -85,B 0,C 180,E1 -26801.188,E2 -26801.188} C_VEL
LIN {X 0,Y 148.322,Z 422.904,A -85,B 0,C 180,E1 -26803.483,E2 -26803.483} C_VEL
LIN {X 0,Y 148.008,Z 423.453,A -85,B 0,C 180,E1 -26806.265,E2 -26806.265} C_VEL
LIN {X 0,Y 146.97,Z 424.632,A -85,B 0,C 180,E1 -26808.972,E2 -26808.972} C_VEL
LIN {X 0,Y 137.429,Z 429.959,A -85,B 0,C 180,E1 -26812.654,E2 -26812.654} C_VEL
LIN {X 0,Y 128.63,Z 433.795,A -85,B 0,C 180,E1 -26816.868,E2 -26816.868} C_VEL
LIN {X 0,Y 123.282,Z 435.618,A -85,B 0,C 180,E1 -26820,E2 -26820} C_VEL
LIN {X 0,Y 118.313,Z 436.852,A -85,B 0,C 180,E1 -26823.405,E2 -26823.405} C_VEL
LIN {X 0,Y 113.406,Z 437.599,A -85,B 0,C 180,E1 -26827.447,E2 -26827.447} C_VEL
LIN {X 0,Y 108.162,Z 437.621,A -85,B 0,C 180,E1 -26832.927,E2 -26832.927} C_VEL
LIN {X 0,Y 103.452,Z 436.388,A -85,B 0,C 180,E1 -26839.857,E2 -26839.857} C_VEL
LIN {X 0,Y 100.46,Z 434.075,A -85,B 0,C 180,E1 -26846.587,E2 -26846.587} C_VEL
LIN {X 0,Y 98.862,Z 432.696,A -85,B 0,C 180,E1 -26849.736,E2 -26849.736} C_VEL
LIN {X 0,Y 95.095,Z 429.765,A -85,B 0,C 180,E1 -26854.863,E2 -26854.863} C_VEL
LIN {X 0,Y 92.03,Z 426.109,A -85,B 0,C 180,E1 -26860.23,E2 -26860.23} C_VEL
LIN {X 0,Y 91.605,Z 423.525,A -85,B 0,C 180,E1 -26863.587,E2 -26863.587} C_VEL
LIN {X 0,Y 92.984,Z 416.501,A -85,B 0,C 180,E1 -26871.213,E2 -26871.213} C_VEL
LIN {X 0,Y 95.268,Z 408.244,A -85,B 0,C 180,E1 -26878.087,E2 -26878.087} C_VEL
LIN {X 0,Y 98.069,Z 399.44,A -85,B 0,C 180,E1 -26883.726,E2 -26883.726} C_VEL
LIN {X 0,Y 101.276,Z 389.619,A -85,B 0,C 180,E1 -26888.634,E2 -26888.634} C_VEL
LIN {X 0,Y 104.615,Z 379.086,A -85,B 0,C 180,E1 -26892.717,E2 -26892.717} C_VEL
LIN {X 0,Y 104.966,Z 377.974,A -85,B 0,C 180,E1 -26893.08,E2 -26893.08} C_VEL
LIN {X 0,Y 103.31,Z 370.019,A -85,B 0,C 180,E1 -26896.393,E2 -26896.393} C_VEL
LIN {X 0,Y 100.749,Z 360.478,A -85,B 0,C 180,E1 -26900.159,E2 -26900.159} C_VEL
LIN {X 0,Y 97.541,Z 350.912,A -85,B 0,C 180,E1 -26903.795,E2 -26903.795} C_VEL
LIN {X 0,Y 94.807,Z 344.523,A -85,B 0,C 180,E1 -26906.281,E2 -26906.281} C_VEL
LIN {X 0,Y 94.406,Z 342.728,A -85,B 0,C 180,E1 -26906.933,E2 -26906.933} C_VEL
LIN {X 0,Y 94.774,Z 342.669,A -85,B 0,C 180,E1 -26910,E2 -26910} C_VEL
LIN {X 0,Y 94.174,Z 342.751,A -85,B 0,C 180,E1 -26918.584,E2 -26918.584} C_VEL
LIN {X 0,Y 94.021,Z 342.769,A -85,B 0,C 180,E1 -26923.655,E2 -26923.655} C_VEL
LIN {X 0,Y 93.692,Z 342.808,A -85,B 0,C 180,E1 -26932.028,E2 -26932.028} C_VEL
LIN {X 0,Y 93.623,Z 342.823,A -85,B 0,C 180,E1 -26936.77,E2 -26936.77} C_VEL
LIN {X 0,Y 93.599,Z 342.826,A -85,B 0,C 180,E1 -26944.316,E2 -26944.316} C_VEL
LIN {X 0,Y 93.539,Z 342.833,A -85,B 0,C 180,E1 -26952.548,E2 -26952.548} C_VEL
LIN {X 0,Y 93.536,Z 342.831,A -85,B 0,C 180,E1 -26958.709,E2 -26958.709} C_VEL
LIN {X 0,Y 93.586,Z 342.821,A -85,B 0,C 180,E1 -26965.697,E2 -26965.697} C_VEL
LIN {X 0,Y 93.669,Z 342.812,A -85,B 0,C 180,E1 -26974.207,E2 -26974.207} C_VEL
LIN {X 0,Y 93.692,Z 342.814,A -85,B 0,C 180,E1 -26977.973,E2 -26977.973} C_VEL
LIN {X 0,Y 94.063,Z 342.766,A -85,B 0,C 180,E1 -26987.048,E2 -26987.048} C_VEL
LIN {X 0,Y 94.166,Z 342.753,A -85,B 0,C 180,E1 -26991.416,E2 -26991.416} C_VEL
LIN {X 0,Y 94.773,Z 342.678,A -85,B 0,C 180,E1 -27000.001,E2 -27000.001} C_VEL
LIN {X 0,Y 94.175,Z 342.753,A -85,B 0,C 180,E1 -27008.584,E2 -27008.584} C_VEL
LIN {X 0,Y 94.025,Z 342.765,A -85,B 0,C 180,E1 -27013.663,E2 -27013.663} C_VEL
LIN {X 0,Y 93.693,Z 342.803,A -85,B 0,C 180,E1 -27022.028,E2 -27022.028} C_VEL
LIN {X 0,Y 93.627,Z 342.789,A -85,B 0,C 180,E1 -27026.769,E2 -27026.769} C_VEL
LIN {X 0,Y 94.081,Z 342.841,A -85,B 0,C 180,E1 -27036.7,E2 -27036.7} C_VEL
LIN {X 0,Y 94.209,Z 343.825,A -85,B 0,C 180,E1 -27038.838,E2 -27038.838} C_VEL
LIN {X 0,Y 95.302,Z 347.282,A -85,B 0,C 180,E1 -27039.841,E2 -27039.841} C_VEL
LIN {X 0,Y 98.525,Z 356.489,A -85,B 0,C 180,E1 -27042.662,E2 -27042.662} C_VEL
LIN {X 0,Y 100.243,Z 362.675,A -85,B 0,C 180,E1 -27044.516,E2 -27044.516} C_VEL
LIN {X 0,Y 100.325,Z 375.146,A -85,B 0,C 180,E1 -27047.807,E2 -27047.807} C_VEL
LIN {X 0,Y 99.95,Z 388.133,A -85,B 0,C 180,E1 -27052.029,E2 -27052.029} C_VEL
LIN {X 0,Y 99.349,Z 399.079,A -85,B 0,C 180,E1 -27056.382,E2 -27056.382} C_VEL
LIN {X 0,Y 98.619,Z 409.115,A -85,B 0,C 180,E1 -27061.247,E2 -27061.247} C_VEL
LIN {X 0,Y 95.913,Z 417.659,A -85,B 0,C 180,E1 -27066.233,E2 -27066.233} C_VEL
LIN {X 0,Y 93.717,Z 426.086,A -85,B 0,C 180,E1 -27072.544,E2 -27072.544} C_VEL
LIN {X 0,Y 92.506,Z 432.79,A -85,B 0,C 180,E1 -27079.051,E2 -27079.051} C_VEL
LIN {X 0,Y 92.345,Z 438.12,A -85,B 0,C 180,E1 -27085.635,E2 -27085.635} C_VEL
LIN {X 0,Y 92.6,Z 440.954,A -85,B 0,C 180,E1 -27090,E2 -27090} C_VEL
LIN {X 0,Y 92.244,Z 443.132,A -85,B 0,C 180,E1 -27094.37,E2 -27094.37} C_VEL
LIN {X 0,Y 92.047,Z 444.827,A -85,B 0,C 180,E1 -27098.784,E2 -27098.784} C_VEL
LIN {X 0,Y 93.151,Z 447.073,A -85,B 0,C 180,E1 -27107.565,E2 -27107.565} C_VEL
LIN {X 0,Y 96.529,Z 447.999,A -85,B 0,C 180,E1 -27115.903,E2 -27115.903} C_VEL
LIN {X 0,Y 102.082,Z 447.637,A -85,B 0,C 180,E1 -27123.42,E2 -27123.42} C_VEL
LIN {X 0,Y 109.237,Z 445.964,A -85,B 0,C 180,E1 -27130.044,E2 -27130.044} C_VEL
LIN {X 0,Y 117.898,Z 442.936,A -85,B 0,C 180,E1 -27135.671,E2 -27135.671} C_VEL
LIN {X 0,Y 127.869,Z 438.501,A -85,B 0,C 180,E1 -27140.307,E2 -27140.307} C_VEL
LIN {X 0,Y 132.638,Z 435.778,A -85,B 0,C 180,E1 -27142.637,E2 -27142.637} C_VEL
LIN {X 0,Y 138.889,Z 431.505,A -85,B 0,C 180,E1 -27146.177,E2 -27146.177} C_VEL
LIN {X 0,Y 140.393,Z 429.886,A -85,B 0,C 180,E1 -27148.323,E2 -27148.323} C_VEL
LIN {X 0,Y 141.73,Z 427.619,A -85,B 0,C 180,E1 -27153.199,E2 -27153.199} C_VEL
LIN {X 0,Y 142.315,Z 426.582,A -85,B 0,C 180,E1 -27156.729,E2 -27156.729} C_VEL
LIN {X 0,Y 142.395,Z 426.273,A -85,B 0,C 180,E1 -27159.788,E2 -27159.788} C_VEL
LIN {X 0,Y 142.209,Z 426.367,A -85,B 0,C 180,E1 -27162.751,E2 -27162.751} C_VEL
LIN {X 0,Y 141.823,Z 426.776,A -85,B 0,C 180,E1 -27165.654,E2 -27165.654} C_VEL
LIN {X 0,Y 141.286,Z 427.224,A -85,B 0,C 180,E1 -27167.065,E2 -27167.065} C_VEL
LIN {X 0,Y 138.551,Z 428.7,A -85,B 0,C 180,E1 -27168.293,E2 -27168.293} C_VEL
LIN {X 0,Y 131.991,Z 431.856,A -85,B 0,C 180,E1 -27170.808,E2 -27170.808} C_VEL
LIN {X 0,Y 125.752,Z 434.304,A -85,B 0,C 180,E1 -27173.582,E2 -27173.582} C_VEL
LIN {X 0,Y 119.661,Z 436.244,A -85,B 0,C 180,E1 -27176.822,E2 -27176.822} C_VEL
LIN {X 0,Y 112.486,Z 437.798,A -85,B 0,C 180,E1 -27181.465,E2 -27181.465} C_VEL
LIN {X 0,Y 105.106,Z 438.354,A -85,B 0,C 180,E1 -27187.685,E2 -27187.685} C_VEL
LIN {X 0,Y 100.778,Z 437.97,A -85,B 0,C 180,E1 -27192.491,E2 -27192.491} C_VEL
LIN {X 0,Y 96.569,Z 436.571,A -85,B 0,C 180,E1 -27198.895,E2 -27198.895} C_VEL
LIN {X 0,Y 93.144,Z 433.647,A -85,B 0,C 180,E1 -27206.918,E2 -27206.918} C_VEL
LIN {X 0,Y 91.515,Z 429.378,A -85,B 0,C 180,E1 -27215.164,E2 -27215.164} C_VEL
LIN {X 0,Y 91.438,Z 425.114,A -85,B 0,C 180,E1 -27221.516,E2 -27221.516} C_VEL
LIN {X 0,Y 91.605,Z 423.525,A -85,B 0,C 180,E1 -27223.587,E2 -27223.587} C_VEL
LIN {X 0,Y 91.4,Z 420.79,A -85,B 0,C 180,E1 -27226.855,E2 -27226.855} C_VEL
LIN {X 0,Y 90.45,Z 417.785,A -85,B 0,C 180,E1 -27230.028,E2 -27230.028} C_VEL
LIN {X 0,Y 88.388,Z 409.917,A -85,B 0,C 180,E1 -27237.302,E2 -27237.302} C_VEL
LIN {X 0,Y 88.881,Z 406.113,A -85,B 0,C 180,E1 -27240.284,E2 -27240.284} C_VEL
LIN {X 0,Y 91.576,Z 398.137,A -85,B 0,C 180,E1 -27245.487,E2 -27245.487} C_VEL
LIN {X 0,Y 95.245,Z 387.562,A -85,B 0,C 180,E1 -27250.815,E2 -27250.815} C_VEL
LIN {X 0,Y 97.92,Z 379.34,A -85,B 0,C 180,E1 -27254.075,E2 -27254.075} C_VEL
LIN {X 0,Y 97.594,Z 376.008,A -85,B 0,C 180,E1 -27255.534,E2 -27255.534} C_VEL
LIN {X 0,Y 95.102,Z 365.578,A -85,B 0,C 180,E1 -27260.155,E2 -27260.155} C_VEL
LIN {X 0,Y 91.754,Z 354.751,A -85,B 0,C 180,E1 -27264.713,E2 -27264.713} C_VEL
LIN {X 0,Y 87.635,Z 343.883,A -85,B 0,C 180,E1 -27269.282,E2 -27269.282} C_VEL
LIN {X 0,Y 87.636,Z 343.56,A -85,B 0,C 180,E1 -27269.426,E2 -27269.426} C_VEL
LIN {X 0,Y 87.083,Z 343.637,A -85,B 0,C 180,E1 -27279.289,E2 -27279.289} C_VEL
LIN {X 0,Y 86.931,Z 343.651,A -85,B 0,C 180,E1 -27284.036,E2 -27284.036} C_VEL
LIN {X 0,Y 86.645,Z 343.692,A -85,B 0,C 180,E1 -27288.932,E2 -27288.932} C_VEL
LIN {X 0,Y 86.585,Z 343.699,A -85,B 0,C 180,E1 -27296.767,E2 -27296.767} C_VEL
LIN {X 0,Y 86.517,Z 343.708,A -85,B 0,C 180,E1 -27305.677,E2 -27305.677} C_VEL
LIN {X 0,Y 86.481,Z 343.712,A -85,B 0,C 180,E1 -27312.997,E2 -27312.997} C_VEL
LIN {X 0,Y 86.458,Z 343.714,A -85,B 0,C 180,E1 -27319.436,E2 -27319.436} C_VEL
LIN {X 0,Y 86.53,Z 343.699,A -85,B 0,C 180,E1 -27325.352,E2 -27325.352} C_VEL
LIN {X 0,Y 86.583,Z 343.693,A -85,B 0,C 180,E1 -27333.237,E2 -27333.237} C_VEL
LIN {X 0,Y 86.632,Z 343.687,A -85,B 0,C 180,E1 -27341.065,E2 -27341.065} C_VEL
LIN {X 0,Y 86.904,Z 343.659,A -85,B 0,C 180,E1 -27346.039,E2 -27346.039} C_VEL
LIN {X 0,Y 87.077,Z 343.633,A -85,B 0,C 180,E1 -27350.711,E2 -27350.711} C_VEL
LIN {X 0,Y 87.703,Z 343.559,A -85,B 0,C 180,E1 -27360.001,E2 -27360.001} C_VEL
LIN {X 0,Y 87.085,Z 343.637,A -85,B 0,C 180,E1 -27369.289,E2 -27369.289} C_VEL
LIN {X 0,Y 86.932,Z 343.649,A -85,B 0,C 180,E1 -27374.037,E2 -27374.037} C_VEL
LIN {X 0,Y 86.646,Z 343.691,A -85,B 0,C 180,E1 -27378.933,E2 -27378.933} C_VEL
LIN {X 0,Y 86.588,Z 343.665,A -85,B 0,C 180,E1 -27386.769,E2 -27386.769} C_VEL
LIN {X 0,Y 86.942,Z 343.654,A -85,B 0,C 180,E1 -27395.915,E2 -27395.915} C_VEL
LIN {X 0,Y 91.142,Z 355.14,A -85,B 0,C 180,E1 -27399.91,E2 -27399.91} C_VEL
LIN {X 0,Y 93.785,Z 364.341,A -85,B 0,C 180,E1 -27402.997,E2 -27402.997} C_VEL
LIN {X 0,Y 93.698,Z 376.224,A -85,B 0,C 180,E1 -27406.49,E2 -27406.49} C_VEL
LIN {X 0,Y 93.138,Z 388.737,A -85,B 0,C 180,E1 -27410.939,E2 -27410.939} C_VEL
LIN {X 0,Y 92.337,Z 400.094,A -85,B 0,C 180,E1 -27415.933,E2 -27415.933} C_VEL
LIN {X 0,Y 91.714,Z 408.085,A -85,B 0,C 180,E1 -27420.126,E2 -27420.126} C_VEL
LIN {X 0,Y 88.985,Z 416.745,A -85,B 0,C 180,E1 -27425.503,E2 -27425.503} C_VEL
LIN {X 0,Y 86.681,Z 425.224,A -85,B 0,C 180,E1 -27432.299,E2 -27432.299} C_VEL
LIN {X 0,Y 85.476,Z 432.001,A -85,B 0,C 180,E1 -27439.339,E2 -27439.339} C_VEL
LIN {X 0,Y 85.338,Z 436.549,A -85,B 0,C 180,E1 -27445.276,E2 -27445.276} C_VEL
LIN {X 0,Y 85.596,Z 439.529,A -85,B 0,C 180,E1 -27450,E2 -27450} C_VEL
LIN {X 0,Y 85.265,Z 441.792,A -85,B 0,C 180,E1 -27454.728,E2 -27454.728} C_VEL
LIN {X 0,Y 85.435,Z 445.021,A -85,B 0,C 180,E1 -27464.288,E2 -27464.288} C_VEL
LIN {X 0,Y 88.005,Z 446.863,A -85,B 0,C 180,E1 -27473.534,E2 -27473.534} C_VEL
LIN {X 0,Y 92.975,Z 447.374,A -85,B 0,C 180,E1 -27481.947,E2 -27481.947} C_VEL
LIN {X 0,Y 99.826,Z 446.588,A -85,B 0,C 180,E1 -27489.318,E2 -27489.318} C_VEL
LIN {X 0,Y 108.301,Z 444.536,A -85,B 0,C 180,E1 -27495.548,E2 -27495.548} C_VEL
LIN {X 0,Y 118.155,Z 441.153,A -85,B 0,C 180,E1 -27500.648,E2 -27500.648} C_VEL
LIN {X 0,Y 123.449,Z 438.911,A -85,B 0,C 180,E1 -27502.848,E2 -27502.848} C_VEL
LIN {X 0,Y 128.371,Z 436.385,A -85,B 0,C 180,E1 -27505.207,E2 -27505.207} C_VEL
LIN {X 0,Y 133.025,Z 433.607,A -85,B 0,C 180,E1 -27507.706,E2 -27507.706} C_VEL
LIN {X 0,Y 134.98,Z 431.399,A -85,B 0,C 180,E1 -27512.056,E2 -27512.056} C_VEL
LIN {X 0,Y 135.752,Z 430.257,A -85,B 0,C 180,E1 -27515.533,E2 -27515.533} C_VEL
LIN {X 0,Y 136.057,Z 429.695,A -85,B 0,C 180,E1 -27518.802,E2 -27518.802} C_VEL
LIN {X 0,Y 135.925,Z 429.561,A -85,B 0,C 180,E1 -27521.926,E2 -27521.926} C_VEL
LIN {X 0,Y 135.516,Z 429.818,A -85,B 0,C 180,E1 -27524.971,E2 -27524.971} C_VEL
LIN {X 0,Y 133.477,Z 430.824,A -85,B 0,C 180,E1 -27526.294,E2 -27526.294} C_VEL
LIN {X 0,Y 123.365,Z 434.802,A -85,B 0,C 180,E1 -27530.159,E2 -27530.159} C_VEL
LIN {X 0,Y 117.16,Z 436.697,A -85,B 0,C 180,E1 -27533.109,E2 -27533.109} C_VEL
LIN {X 0,Y 111.272,Z 437.999,A -85,B 0,C 180,E1 -27536.378,E2 -27536.378} C_VEL
LIN {X 0,Y 105.422,Z 438.823,A -85,B 0,C 180,E1 -27540.287,E2 -27540.287} C_VEL
LIN {X 0,Y 98.899,Z 438.95,A -85,B 0,C 180,E1 -27545.796,E2 -27545.796} C_VEL
LIN {X 0,Y 92.533,Z 437.858,A -85,B 0,C 180,E1 -27553.17,E2 -27553.17} C_VEL
LIN {X 0,Y 89.117,Z 436.292,A -85,B 0,C 180,E1 -27558.851,E2 -27558.851} C_VEL
LIN {X 0,Y 86.139,Z 433.51,A -85,B 0,C 180,E1 -27566.17,E2 -27566.17} C_VEL
LIN {X 0,Y 84.553,Z 429.722,A -85,B 0,C 180,E1 -27573.778,E2 -27573.778} C_VEL
LIN {X 0,Y 84.379,Z 424.609,A -85,B 0,C 180,E1 -27581.783,E2 -27581.783} C_VEL
LIN {X 0,Y 85.532,Z 417.942,A -85,B 0,C 180,E1 -27589.846,E2 -27589.846} C_VEL
LIN {X 0,Y 87.409,Z 410.851,A -85,B 0,C 180,E1 -27596.562,E2 -27596.562} C_VEL
LIN {X 0,Y 88.881,Z 406.113,A -85,B 0,C 180,E1 -27600.284,E2 -27600.284} C_VEL
LIN {X 0,Y 89.497,Z 402.195,A -85,B 0,C 180,E1 -27603.103,E2 -27603.103} C_VEL
LIN {X 0,Y 89.07,Z 395.307,A -85,B 0,C 180,E1 -27607.687,E2 -27607.687} C_VEL
LIN {X 0,Y 88.971,Z 387.901,A -85,B 0,C 180,E1 -27611.965,E2 -27611.965} C_VEL
LIN {X 0,Y 90.046,Z 383.17,A -85,B 0,C 180,E1 -27614.144,E2 -27614.144} C_VEL
LIN {X 0,Y 91.165,Z 379.817,A -85,B 0,C 180,E1 -27615.49,E2 -27615.49} C_VEL
LIN {X 0,Y 89.209,Z 370.146,A -85,B 0,C 180,E1 -27620.217,E2 -27620.217} C_VEL
LIN {X 0,Y 86.586,Z 360.61,A -85,B 0,C 180,E1 -27624.732,E2 -27624.732} C_VEL
LIN {X 0,Y 83.164,Z 351.054,A -85,B 0,C 180,E1 -27629.333,E2 -27629.333} C_VEL
LIN {X 0,Y 82.135,Z 348.262,A -85,B 0,C 180,E1 -27630.613,E2 -27630.613} C_VEL
LIN {X 0,Y 80.819,Z 346.168,A -85,B 0,C 180,E1 -27631.869,E2 -27631.869} C_VEL
LIN {X 0,Y 80.302,Z 344.477,A -85,B 0,C 180,E1 -27632.665,E2 -27632.665} C_VEL
LIN {X 0,Y 79.967,Z 344.524,A -85,B 0,C 180,E1 -27640.124,E2 -27640.124} C_VEL
LIN {X 0,Y 79.744,Z 344.547,A -85,B 0,C 180,E1 -27645.331,E2 -27645.331} C_VEL
LIN {X 0,Y 79.513,Z 344.576,A -85,B 0,C 180,E1 -27650.705,E2 -27650.705} C_VEL
LIN {X 0,Y 79.483,Z 344.583,A -85,B 0,C 180,E1 -27657.847,E2 -27657.847} C_VEL
LIN {X 0,Y 79.385,Z 344.592,A -85,B 0,C 180,E1 -27662.086,E2 -27662.086} C_VEL
LIN {X 0,Y 79.373,Z 344.59,A -85,B 0,C 180,E1 -27668.303,E2 -27668.303} C_VEL
LIN {X 0,Y 79.41,Z 344.589,A -85,B 0,C 180,E1 -27675.075,E2 -27675.075} C_VEL
LIN {X 0,Y 79.386,Z 344.594,A -85,B 0,C 180,E1 -27682.823,E2 -27682.823} C_VEL
LIN {X 0,Y 79.376,Z 344.597,A -85,B 0,C 180,E1 -27687.911,E2 -27687.911} C_VEL
LIN {X 0,Y 79.524,Z 344.572,A -85,B 0,C 180,E1 -27693.777,E2 -27693.777} C_VEL
LIN {X 0,Y 79.506,Z 344.578,A -85,B 0,C 180,E1 -27699.294,E2 -27699.294} C_VEL
LIN {X 0,Y 79.81,Z 344.544,A -85,B 0,C 180,E1 -27705.617,E2 -27705.617} C_VEL
LIN {X 0,Y 79.957,Z 344.518,A -85,B 0,C 180,E1 -27709.876,E2 -27709.876} C_VEL
LIN {X 0,Y 80.632,Z 344.439,A -85,B 0,C 180,E1 -27720.001,E2 -27720.001} C_VEL
LIN {X 0,Y 79.968,Z 344.524,A -85,B 0,C 180,E1 -27730.124,E2 -27730.124} C_VEL
LIN {X 0,Y 79.745,Z 344.547,A -85,B 0,C 180,E1 -27735.332,E2 -27735.332} C_VEL
LIN {X 0,Y 79.514,Z 344.575,A -85,B 0,C 180,E1 -27740.705,E2 -27740.705} C_VEL
LIN {X 0,Y 79.52,Z 344.547,A -85,B 0,C 180,E1 -27747.895,E2 -27747.895} C_VEL
LIN {X 0,Y 79.592,Z 344.648,A -85,B 0,C 180,E1 -27752.554,E2 -27752.554} C_VEL
LIN {X 0,Y 80.702,Z 347.421,A -85,B 0,C 180,E1 -27753.724,E2 -27753.724} C_VEL
LIN {X 0,Y 82.135,Z 349.518,A -85,B 0,C 180,E1 -27754.906,E2 -27754.906} C_VEL
LIN {X 0,Y 85.123,Z 358.09,A -85,B 0,C 180,E1 -27758.332,E2 -27758.332} C_VEL
LIN {X 0,Y 87.106,Z 365.107,A -85,B 0,C 180,E1 -27761.04,E2 -27761.04} C_VEL
LIN {X 0,Y 87.369,Z 369.535,A -85,B 0,C 180,E1 -27762.48,E2 -27762.48} C_VEL
LIN {X 0,Y 86.786,Z 382.101,A -85,B 0,C 180,E1 -27766.789,E2 -27766.789} C_VEL
LIN {X 0,Y 85.984,Z 393.193,A -85,B 0,C 180,E1 -27771.447,E2 -27771.447} C_VEL
LIN {X 0,Y 85.115,Z 403.05,A -85,B 0,C 180,E1 -27776.479,E2 -27776.479} C_VEL
LIN {X 0,Y 84.429,Z 409.025,A -85,B 0,C 180,E1 -27780.036,E2 -27780.036} C_VEL
LIN {X 0,Y 81.603,Z 417.361,A -85,B 0,C 180,E1 -27785.852,E2 -27785.852} C_VEL
LIN {X 0,Y 79.39,Z 425.554,A -85,B 0,C 180,E1 -27793.279,E2 -27793.279} C_VEL
LIN {X 0,Y 78.401,Z 431.679,A -85,B 0,C 180,E1 -27800.425,E2 -27800.425} C_VEL
LIN {X 0,Y 78.421,Z 436.503,A -85,B 0,C 180,E1 -27807.432,E2 -27807.432} C_VEL
LIN {X 0,Y 78.594,Z 437.986,A -85,B 0,C 180,E1 -27810,E2 -27810} C_VEL
LIN {X 0,Y 78.296,Z 440.43,A -85,B 0,C 180,E1 -27815.15,E2 -27815.15} C_VEL
LIN {X 0,Y 78.189,Z 442.358,A -85,B 0,C 180,E1 -27820.357,E2 -27820.357} C_VEL
LIN {X 0,Y 79.765,Z 445.058,A -85,B 0,C 180,E1 -27830.637,E2 -27830.637} C_VEL
LIN {X 0,Y 83.984,Z 446.467,A -85,B 0,C 180,E1 -27840.139,E2 -27840.139} C_VEL
LIN {X 0,Y 90.549,Z 446.619,A -85,B 0,C 180,E1 -27848.384,E2 -27848.384} C_VEL
LIN {X 0,Y 98.767,Z 445.48,A -85,B 0,C 180,E1 -27855.364,E2 -27855.364} C_VEL
LIN {X 0,Y 108.47,Z 443.035,A -85,B 0,C 180,E1 -27861.033,E2 -27861.033} C_VEL
LIN {X 0,Y 119.274,Z 439.271,A -85,B 0,C 180,E1 -27865.582,E2 -27865.582} C_VEL
LIN {X 0,Y 124.373,Z 436.924,A -85,B 0,C 180,E1 -27867.954,E2 -27867.954} C_VEL
LIN {X 0,Y 127.42,Z 435.137,A -85,B 0,C 180,E1 -27870.237,E2 -27870.237} C_VEL
LIN {X 0,Y 128.858,Z 433.652,A -85,B 0,C 180,E1 -27874.13,E2 -27874.13} C_VEL
LIN {X 0,Y 129.474,Z 432.821,A -85,B 0,C 180,E1 -27877.668,E2 -27877.668} C_VEL
LIN {X 0,Y 129.457,Z 432.517,A -85,B 0,C 180,E1 -27880.99,E2 -27880.99} C_VEL
LIN {X 0,Y 128.542,Z 432.803,A -85,B 0,C 180,E1 -27884.134,E2 -27884.134} C_VEL
LIN {X 0,Y 121.499,Z 435.341,A -85,B 0,C 180,E1 -27886.621,E2 -27886.621} C_VEL
LIN {X 0,Y 114.313,Z 437.393,A -85,B 0,C 180,E1 -27889.638,E2 -27889.638} C_VEL
LIN {X 0,Y 106.015,Z 438.984,A -85,B 0,C 180,E1 -27893.931,E2 -27893.931} C_VEL
LIN {X 0,Y 97.009,Z 439.655,A -85,B 0,C 180,E1 -27899.999,E2 -27899.999} C_VEL
LIN {X 0,Y 91.677,Z 439.331,A -85,B 0,C 180,E1 -27904.732,E2 -27904.732} C_VEL
LIN {X 0,Y 86.021,Z 438.071,A -85,B 0,C 180,E1 -27911.358,E2 -27911.358} C_VEL
LIN {X 0,Y 80.983,Z 435.304,A -85,B 0,C 180,E1 -27920.312,E2 -27920.312} C_VEL
LIN {X 0,Y 78.079,Z 431.251,A -85,B 0,C 180,E1 -27929.67,E2 -27929.67} C_VEL
LIN {X 0,Y 77.209,Z 425.672,A -85,B 0,C 180,E1 -27939.581,E2 -27939.581} C_VEL
LIN {X 0,Y 77.719,Z 420.864,A -85,B 0,C 180,E1 -27946.338,E2 -27946.338} C_VEL
LIN {X 0,Y 79.501,Z 413.631,A -85,B 0,C 180,E1 -27954.45,E2 -27954.45} C_VEL
LIN {X 0,Y 82.01,Z 405.69,A -85,B 0,C 180,E1 -27961.374,E2 -27961.374} C_VEL
LIN {X 0,Y 85.099,Z 396.945,A -85,B 0,C 180,E1 -27967.304,E2 -27967.304} C_VEL
LIN {X 0,Y 89.27,Z 385.366,A -85,B 0,C 180,E1 -27973.22,E2 -27973.22} C_VEL
LIN {X 0,Y 90.046,Z 383.17,A -85,B 0,C 180,E1 -27974.144,E2 -27974.144} C_VEL
LIN {X 0,Y 90.187,Z 380.65,A -85,B 0,C 180,E1 -27975.337,E2 -27975.337} C_VEL
LIN {X 0,Y 89.201,Z 378.365,A -85,B 0,C 180,E1 -27976.668,E2 -27976.668} C_VEL
LIN {X 0,Y 87.227,Z 375.988,A -85,B 0,C 180,E1 -27978.322,E2 -27978.322} C_VEL
LIN {X 0,Y 82.768,Z 371.023,A -85,B 0,C 180,E1 -27982.02,E2 -27982.02} C_VEL
LIN {X 0,Y 81.886,Z 368.963,A -85,B 0,C 180,E1 -27983.236,E2 -27983.236} C_VEL
LIN {X 0,Y 79.332,Z 360.008,A -85,B 0,C 180,E1 -27987.952,E2 -27987.952} C_VEL
LIN {X 0,Y 76.763,Z 352.639,A -85,B 0,C 180,E1 -27991.9,E2 -27991.9} C_VEL
LIN {X 0,Y 74.966,Z 349.304,A -85,B 0,C 180,E1 -27994.03,E2 -27994.03} C_VEL
LIN {X 0,Y 73.621,Z 347.434,A -85,B 0,C 180,E1 -27995.478,E2 -27995.478} C_VEL
LIN {X 0,Y 72.959,Z 345.394,A -85,B 0,C 180,E1 -27996.568,E2 -27996.568} C_VEL
LIN {X 0,Y 72.858,Z 345.41,A -85,B 0,C 180,E1 -28001.123,E2 -28001.123} C_VEL
LIN {X 0,Y 72.573,Z 345.444,A -85,B 0,C 180,E1 -28006.889,E2 -28006.889} C_VEL
LIN {X 0,Y 72.394,Z 345.46,A -85,B 0,C 180,E1 -28012.85,E2 -28012.85} C_VEL
LIN {X 0,Y 72.376,Z 345.464,A -85,B 0,C 180,E1 -28019.083,E2 -28019.083} C_VEL
LIN {X 0,Y 72.3,Z 345.478,A -85,B 0,C 180,E1 -28025.679,E2 -28025.679} C_VEL
LIN {X 0,Y 72.261,Z 345.484,A -85,B 0,C 180,E1 -28032.907,E2 -28032.907} C_VEL
LIN {X 0,Y 72.295,Z 345.48,A -85,B 0,C 180,E1 -28041.051,E2 -28041.051} C_VEL
LIN {X 0,Y 72.293,Z 345.472,A -85,B 0,C 180,E1 -28044.319,E2 -28044.319} C_VEL
LIN {X 0,Y 72.358,Z 345.469,A -85,B 0,C 180,E1 -28050.946,E2 -28050.946} C_VEL
LIN {X 0,Y 72.39,Z 345.468,A -85,B 0,C 180,E1 -28057.149,E2 -28057.149} C_VEL
LIN {X 0,Y 72.709,Z 345.429,A -85,B 0,C 180,E1 -28065.15,E2 -28065.15} C_VEL
LIN {X 0,Y 72.847,Z 345.403,A -85,B 0,C 180,E1 -28068.876,E2 -28068.876} C_VEL
LIN {X 0,Y 73.56,Z 345.32,A -85,B 0,C 180,E1 -28080.001,E2 -28080.001} C_VEL
LIN {X 0,Y 72.859,Z 345.408,A -85,B 0,C 180,E1 -28091.124,E2 -28091.124} C_VEL
LIN {X 0,Y 72.575,Z 345.444,A -85,B 0,C 180,E1 -28096.89,E2 -28096.89} C_VEL
LIN {X 0,Y 72.495,Z 345.419,A -85,B 0,C 180,E1 -28107.42,E2 -28107.42} C_VEL
LIN {X 0,Y 72.479,Z 345.625,A -85,B 0,C 180,E1 -28108.648,E2 -28108.648} C_VEL
LIN {X 0,Y 73.683,Z 348.636,A -85,B 0,C 180,E1 -28110.188,E2 -28110.188} C_VEL
LIN {X 0,Y 74.825,Z 350.365,A -85,B 0,C 180,E1 -28111.301,E2 -28111.301} C_VEL
LIN {X 0,Y 77.155,Z 354.551,A -85,B 0,C 180,E1 -28113.718,E2 -28113.718} C_VEL
LIN {X 0,Y 80.429,Z 365.796,A -85,B 0,C 180,E1 -28118.704,E2 -28118.704} C_VEL
LIN {X 0,Y 80.987,Z 368.601,A -85,B 0,C 180,E1 -28119.888,E2 -28119.888} C_VEL
LIN {X 0,Y 80.211,Z 381.12,A -85,B 0,C 180,E1 -28124.504,E2 -28124.504} C_VEL
LIN {X 0,Y 79.34,Z 391.574,A -85,B 0,C 180,E1 -28129.21,E2 -28129.21} C_VEL
LIN {X 0,Y 78.25,Z 402.064,A -85,B 0,C 180,E1 -28134.92,E2 -28134.92} C_VEL
LIN {X 0,Y 77.682,Z 407.857,A -85,B 0,C 180,E1 -28138.654,E2 -28138.654} C_VEL
LIN {X 0,Y 74.706,Z 416.291,A -85,B 0,C 180,E1 -28144.954,E2 -28144.954} C_VEL
LIN {X 0,Y 72.363,Z 424.587,A -85,B 0,C 180,E1 -28153.06,E2 -28153.06} C_VEL
LIN {X 0,Y 71.359,Z 431.353,A -85,B 0,C 180,E1 -28161.748,E2 -28161.748} C_VEL
LIN {X 0,Y 71.591,Z 436.402,A -85,B 0,C 180,E1 -28170,E2 -28170} C_VEL
LIN {X 0,Y 71.565,Z 437.796,A -85,B 0,C 180,E1 -28172.815,E2 -28172.815} C_VEL
LIN {X 0,Y 71.306,Z 440.992,A -85,B 0,C 180,E1 -28181.369,E2 -28181.369} C_VEL
LIN {X 0,Y 73.19,Z 443.981,A -85,B 0,C 180,E1 -28192.588,E2 -28192.588} C_VEL
LIN {X 0,Y 77.929,Z 445.625,A -85,B 0,C 180,E1 -28202.759,E2 -28202.759} C_VEL
LIN {X 0,Y 85.091,Z 446.012,A -85,B 0,C 180,E1 -28211.358,E2 -28211.358} C_VEL
LIN {X 0,Y 93.898,Z 445.137,A -85,B 0,C 180,E1 -28218.459,E2 -28218.459} C_VEL
LIN {X 0,Y 104.148,Z 443.028,A -85,B 0,C 180,E1 -28224.074,E2 -28224.074} C_VEL
LIN {X 0,Y 115.381,Z 439.593,A -85,B 0,C 180,E1 -28228.514,E2 -28228.514} C_VEL
LIN {X 0,Y 118.062,Z 438.524,A -85,B 0,C 180,E1 -28229.674,E2 -28229.674} C_VEL
LIN {X 0,Y 120.405,Z 437.478,A -85,B 0,C 180,E1 -28231.111,E2 -28231.111} C_VEL
LIN {X 0,Y 121.533,Z 436.79,A -85,B 0,C 180,E1 -28232.443,E2 -28232.443} C_VEL
LIN {X 0,Y 122.575,Z 435.663,A -85,B 0,C 180,E1 -28236.547,E2 -28236.547} C_VEL
LIN {X 0,Y 122.821,Z 435.188,A -85,B 0,C 180,E1 -28239.92,E2 -28239.92} C_VEL
LIN {X 0,Y 122.565,Z 435.145,A -85,B 0,C 180,E1 -28241.616,E2 -28241.616} C_VEL
LIN {X 0,Y 120.112,Z 435.89,A -85,B 0,C 180,E1 -28242.988,E2 -28242.988} C_VEL
LIN {X 0,Y 112.997,Z 437.834,A -85,B 0,C 180,E1 -28245.594,E2 -28245.594} C_VEL
LIN {X 0,Y 106.199,Z 439.204,A -85,B 0,C 180,E1 -28248.548,E2 -28248.548} C_VEL
LIN {X 0,Y 99.324,Z 440.055,A -85,B 0,C 180,E1 -28252.148,E2 -28252.148} C_VEL
LIN {X 0,Y 91.464,Z 440.256,A -85,B 0,C 180,E1 -28257.339,E2 -28257.339} C_VEL
LIN {X 0,Y 83.219,Z 439.279,A -85,B 0,C 180,E1 -28264.844,E2 -28264.844} C_VEL
LIN {X 0,Y 78.659,Z 437.826,A -85,B 0,C 180,E1 -28270.63,E2 -28270.63} C_VEL
LIN {X 0,Y 74.214,Z 435.165,A -85,B 0,C 180,E1 -28278.738,E2 -28278.738} C_VEL
LIN {X 0,Y 71.351,Z 431.498,A -85,B 0,C 180,E1 -28287.563,E2 -28287.563} C_VEL
LIN {X 0,Y 70.127,Z 425.604,A -85,B 0,C 180,E1 -28298.781,E2 -28298.781} C_VEL
LIN {X 0,Y 70.974,Z 418.93,A -85,B 0,C 180,E1 -28308.541,E2 -28308.541} C_VEL
LIN {X 0,Y 73.293,Z 410.723,A -85,B 0,C 180,E1 -28317.764,E2 -28317.764} C_VEL
LIN {X 0,Y 76.271,Z 402.2,A -85,B 0,C 180,E1 -28325.031,E2 -28325.031} C_VEL
LIN {X 0,Y 79.753,Z 392.851,A -85,B 0,C 180,E1 -28331.085,E2 -28331.085} C_VEL
LIN {X 0,Y 83.546,Z 382.823,A -85,B 0,C 180,E1 -28336.007,E2 -28336.007} C_VEL
LIN {X 0,Y 84.113,Z 381.175,A -85,B 0,C 180,E1 -28336.716,E2 -28336.716} C_VEL
LIN {X 0,Y 84.004,Z 378.821,A -85,B 0,C 180,E1 -28337.927,E2 -28337.927} C_VEL
LIN {X 0,Y 81.886,Z 368.963,A -85,B 0,C 180,E1 -28343.236,E2 -28343.236} C_VEL
LIN {X 0,Y 80.098,Z 364.653,A -85,B 0,C 180,E1 -28345.807,E2 -28345.807} C_VEL
LIN {X 0,Y 77.414,Z 360.907,A -85,B 0,C 180,E1 -28348.556,E2 -28348.556} C_VEL
LIN {X 0,Y 71.042,Z 354.255,A -85,B 0,C 180,E1 -28354.663,E2 -28354.663} C_VEL
LIN {X 0,Y 67.141,Z 349.552,A -85,B 0,C 180,E1 -28359.129,E2 -28359.129} C_VEL
LIN {X 0,Y 65.777,Z 346.292,A -85,B 0,C 180,E1 -28361.557,E2 -28361.557} C_VEL
LIN {X 0,Y 65.38,Z 346.341,A -85,B 0,C 180,E1 -28368.813,E2 -28368.813} C_VEL
LIN {X 0,Y 65.239,Z 346.358,A -85,B 0,C 180,E1 -28375.525,E2 -28375.525} C_VEL
LIN {X 0,Y 65.198,Z 346.36,A -85,B 0,C 180,E1 -28382.614,E2 -28382.614} C_VEL
LIN {X 0,Y 65.193,Z 346.362,A -85,B 0,C 180,E1 -28391.009,E2 -28391.009} C_VEL
LIN {X 0,Y 65.208,Z 346.361,A -85,B 0,C 180,E1 -28399.71,E2 -28399.71} C_VEL
LIN {X 0,Y 65.241,Z 346.358,A -85,B 0,C 180,E1 -28409.519,E2 -28409.519} C_VEL
LIN {X 0,Y 65.228,Z 346.354,A -85,B 0,C 180,E1 -28414.471,E2 -28414.471} C_VEL
LIN {X 0,Y 65.608,Z 346.312,A -85,B 0,C 180,E1 -28424.6,E2 -28424.6} C_VEL
LIN {X 0,Y 65.744,Z 346.291,A -85,B 0,C 180,E1 -28427.656,E2 -28427.656} C_VEL
LIN {X 0,Y 66.485,Z 346.202,A -85,B 0,C 180,E1 -28440.001,E2 -28440.001} C_VEL
LIN {X 0,Y 65.756,Z 346.289,A -85,B 0,C 180,E1 -28452.344,E2 -28452.344} C_VEL
LIN {X 0,Y 65.382,Z 346.34,A -85,B 0,C 180,E1 -28458.813,E2 -28458.813} C_VEL
LIN {X 0,Y 65.375,Z 346.315,A -85,B 0,C 180,E1 -28463.565,E2 -28463.565} C_VEL
LIN {X 0,Y 66.274,Z 348.945,A -85,B 0,C 180,E1 -28465.099,E2 -28465.099} C_VEL
LIN {X 0,Y 67.812,Z 351.171,A -85,B 0,C 180,E1 -28467.021,E2 -28467.021} C_VEL
LIN {X 0,Y 71.75,Z 358.9,A -85,B 0,C 180,E1 -28472.183,E2 -28472.183} C_VEL
LIN {X 0,Y 74.327,Z 368.629,A -85,B 0,C 180,E1 -28477.073,E2 -28477.073} C_VEL
LIN {X 0,Y 74.633,Z 371.299,A -85,B 0,C 180,E1 -28478.255,E2 -28478.255} C_VEL
LIN {X 0,Y 73.504,Z 383.336,A -85,B 0,C 180,E1 -28483.275,E2 -28483.275} C_VEL
LIN {X 0,Y 72.254,Z 394.637,A -85,B 0,C 180,E1 -28489.147,E2 -28489.147} C_VEL
LIN {X 0,Y 71.044,Z 404.399,A -85,B 0,C 180,E1 -28495.332,E2 -28495.332} C_VEL
LIN {X 0,Y 70.285,Z 408.533,A -85,B 0,C 180,E1 -28498.334,E2 -28498.334} C_VEL
LIN {X 0,Y 67.277,Z 416.755,A -85,B 0,C 180,E1 -28505.301,E2 -28505.301} C_VEL
LIN {X 0,Y 65.074,Z 424.797,A -85,B 0,C 180,E1 -28514.336,E2 -28514.336} C_VEL
LIN {X 0,Y 64.374,Z 431.202,A -85,B 0,C 180,E1 -28523.732,E2 -28523.732} C_VEL
LIN {X 0,Y 64.602,Z 434.694,A -85,B 0,C 180,E1 -28530,E2 -28530} C_VEL
LIN {X 0,Y 64.657,Z 436.153,A -85,B 0,C 180,E1 -28533.116,E2 -28533.116} C_VEL
LIN {X 0,Y 64.458,Z 439.586,A -85,B 0,C 180,E1 -28542.596,E2 -28542.596} C_VEL
LIN {X 0,Y 66.746,Z 442.793,A -85,B 0,C 180,E1 -28554.909,E2 -28554.909} C_VEL
LIN {X 0,Y 72.076,Z 444.694,A -85,B 0,C 180,E1 -28565.807,E2 -28565.807} C_VEL
LIN {X 0,Y 79.894,Z 445.375,A -85,B 0,C 180,E1 -28574.728,E2 -28574.728} C_VEL
LIN {X 0,Y 89.336,Z 444.787,A -85,B 0,C 180,E1 -28581.878,E2 -28581.878} C_VEL
LIN {X 0,Y 100.148,Z 442.943,A -85,B 0,C 180,E1 -28587.365,E2 -28587.365} C_VEL
LIN {X 0,Y 111.802,Z 439.841,A -85,B 0,C 180,E1 -28591.65,E2 -28591.65} C_VEL
LIN {X 0,Y 113.997,Z 439.086,A -85,B 0,C 180,E1 -28592.691,E2 -28592.691} C_VEL
LIN {X 0,Y 115.221,Z 438.365,A -85,B 0,C 180,E1 -28594.724,E2 -28594.724} C_VEL
LIN {X 0,Y 115.93,Z 437.59,A -85,B 0,C 180,E1 -28598.67,E2 -28598.67} C_VEL
LIN {X 0,Y 115.455,Z 437.556,A -85,B 0,C 180,E1 -28600.439,E2 -28600.439} C_VEL
LIN {X 0,Y 104.511,Z 439.82,A -85,B 0,C 180,E1 -28604.396,E2 -28604.396} C_VEL
LIN {X 0,Y 92.748,Z 440.916,A -85,B 0,C 180,E1 -28610.093,E2 -28610.093} C_VEL
LIN {X 0,Y 84.597,Z 440.678,A -85,B 0,C 180,E1 -28615.502,E2 -28615.502} C_VEL
LIN {X 0,Y 77.355,Z 439.514,A -85,B 0,C 180,E1 -28621.991,E2 -28621.991} C_VEL
LIN {X 0,Y 70.206,Z 436.818,A -85,B 0,C 180,E1 -28631.549,E2 -28631.549} C_VEL
LIN {X 0,Y 65.565,Z 432.966,A -85,B 0,C 180,E1 -28642.031,E2 -28642.031} C_VEL
LIN {X 0,Y 63.269,Z 427.627,A -85,B 0,C 180,E1 -28653.738,E2 -28653.738} C_VEL
LIN {X 0,Y 63.399,Z 420.959,A -85,B 0,C 180,E1 -28665.298,E2 -28665.298} C_VEL
LIN {X 0,Y 64.933,Z 414.54,A -85,B 0,C 180,E1 -28674.01,E2 -28674.01} C_VEL
LIN {X 0,Y 67.523,Z 406.842,A -85,B 0,C 180,E1 -28682.213,E2 -28682.213} C_VEL
LIN {X 0,Y 71.191,Z 397.431,A -85,B 0,C 180,E1 -28689.786,E2 -28689.786} C_VEL
LIN {X 0,Y 75.856,Z 385.835,A -85,B 0,C 180,E1 -28696.607,E2 -28696.607} C_VEL
LIN {X 0,Y 77.422,Z 381.099,A -85,B 0,C 180,E1 -28698.878,E2 -28698.878} C_VEL
LIN {X 0,Y 75.591,Z 371.793,A -85,B 0,C 180,E1 -28704.424,E2 -28704.424} C_VEL
LIN {X 0,Y 73.637,Z 364.187,A -85,B 0,C 180,E1 -28708.897,E2 -28708.897} C_VEL
LIN {X 0,Y 71.138,Z 356.417,A -85,B 0,C 180,E1 -28713.668,E2 -28713.668} C_VEL
LIN {X 0,Y 67.97,Z 350.473,A -85,B 0,C 180,E1 -28718.174,E2 -28718.174} C_VEL
LIN {X 0,Y 67.141,Z 349.552,A -85,B 0,C 180,E1 -28719.129,E2 -28719.129} C_VEL
LIN {X 0,Y 65.412,Z 347.773,A -85,B 0,C 180,E1 -28721.588,E2 -28721.588} C_VEL
LIN {X 0,Y 62.814,Z 346.82,A -85,B 0,C 180,E1 -28726.121,E2 -28726.121} C_VEL
LIN {X 0,Y 58.149,Z 347.24,A -85,B 0,C 180,E1 -28743.095,E2 -28743.095} C_VEL
LIN {X 0,Y 58.036,Z 347.249,A -85,B 0,C 180,E1 -28747.211,E2 -28747.211} C_VEL
LIN {X 0,Y 58.019,Z 347.249,A -85,B 0,C 180,E1 -28756.619,E2 -28756.619} C_VEL
LIN {X 0,Y 58.026,Z 347.253,A -85,B 0,C 180,E1 -28762.73,E2 -28762.73} C_VEL
LIN {X 0,Y 58.139,Z 347.239,A -85,B 0,C 180,E1 -28771.085,E2 -28771.085} C_VEL
LIN {X 0,Y 58.503,Z 347.196,A -85,B 0,C 180,E1 -28783.956,E2 -28783.956} C_VEL
LIN {X 0,Y 58.794,Z 347.162,A -85,B 0,C 180,E1 -28793.136,E2 -28793.136} C_VEL
LIN {X 0,Y 59.376,Z 347.086,A -85,B 0,C 180,E1 -28800.001,E2 -28800.001} C_VEL
LIN {X 0,Y 58.797,Z 347.154,A -85,B 0,C 180,E1 -28806.866,E2 -28806.866} C_VEL
LIN {X 0,Y 58.497,Z 347.195,A -85,B 0,C 180,E1 -28816.025,E2 -28816.025} C_VEL
LIN {X 0,Y 58.44,Z 347.407,A -85,B 0,C 180,E1 -28817.268,E2 -28817.268} C_VEL
LIN {X 0,Y 59.343,Z 350.078,A -85,B 0,C 180,E1 -28819.344,E2 -28819.344} C_VEL
LIN {X 0,Y 60.932,Z 352.229,A -85,B 0,C 180,E1 -28821.794,E2 -28821.794} C_VEL
LIN {X 0,Y 63.649,Z 357.501,A -85,B 0,C 180,E1 -28826.212,E2 -28826.212} C_VEL
LIN {X 0,Y 66.206,Z 362.782,A -85,B 0,C 180,E1 -28830.281,E2 -28830.281} C_VEL
LIN {X 0,Y 68.339,Z 372.126,A -85,B 0,C 180,E1 -28835.678,E2 -28835.678} C_VEL
LIN {X 0,Y 66.786,Z 385.07,A -85,B 0,C 180,E1 -28841.736,E2 -28841.736} C_VEL
LIN {X 0,Y 65.315,Z 395.989,A -85,B 0,C 180,E1 -28848.133,E2 -28848.133} C_VEL
LIN {X 0,Y 64,Z 405.227,A -85,B 0,C 180,E1 -28854.794,E2 -28854.794} C_VEL
LIN {X 0,Y 62.911,Z 409.1,A -85,B 0,C 180,E1 -28857.951,E2 -28857.951} C_VEL
LIN {X 0,Y 59.441,Z 418.469,A -85,B 0,C 180,E1 -28867.402,E2 -28867.402} C_VEL
LIN {X 0,Y 57.739,Z 425.484,A -85,B 0,C 180,E1 -28876.849,E2 -28876.849} C_VEL
LIN {X 0,Y 57.461,Z 431.138,A -85,B 0,C 180,E1 -28886.494,E2 -28886.494} C_VEL
LIN {X 0,Y 57.772,Z 434.496,A -85,B 0,C 180,E1 -28893.487,E2 -28893.487} C_VEL
LIN {X 0,Y 57.681,Z 438.097,A -85,B 0,C 180,E1 -28904.104,E2 -28904.104} C_VEL
LIN {X 0,Y 60.45,Z 441.57,A -85,B 0,C 180,E1 -28917.713,E2 -28917.713} C_VEL
LIN {X 0,Y 66.469,Z 443.724,A -85,B 0,C 180,E1 -28929.376,E2 -28929.376} C_VEL
LIN {X 0,Y 75.013,Z 444.635,A -85,B 0,C 180,E1 -28938.549,E2 -28938.549} C_VEL
LIN {X 0,Y 85.136,Z 444.326,A -85,B 0,C 180,E1 -28945.64,E2 -28945.64} C_VEL
LIN {X 0,Y 96.508,Z 442.816,A -85,B 0,C 180,E1 -28950.913,E2 -28950.913} C_VEL
LIN {X 0,Y 102.522,Z 441.597,A -85,B 0,C 180,E1 -28953.021,E2 -28953.021} C_VEL
LIN {X 0,Y 108.304,Z 440.068,A -85,B 0,C 180,E1 -28955.297,E2 -28955.297} C_VEL
LIN {X 0,Y 108.802,Z 439.681,A -85,B 0,C 180,E1 -28957.196,E2 -28957.196} C_VEL
LIN {X 0,Y 107.959,Z 439.686,A -85,B 0,C 180,E1 -28958.592,E2 -28958.592} C_VEL
LIN {X 0,Y 95.432,Z 441.337,A -85,B 0,C 180,E1 -28963.212,E2 -28963.212} C_VEL
LIN {X 0,Y 86.313,Z 441.569,A -85,B 0,C 180,E1 -28967.717,E2 -28967.717} C_VEL
LIN {X 0,Y 76.087,Z 440.639,A -85,B 0,C 180,E1 -28974.699,E2 -28974.699} C_VEL
LIN {X 0,Y 70.281,Z 439.291,A -85,B 0,C 180,E1 -28980.208,E2 -28980.208} C_VEL
LIN {X 0,Y 63.979,Z 436.734,A -85,B 0,C 180,E1 -28988.644,E2 -28988.644} C_VEL
LIN {X 0,Y 58.495,Z 432.175,A -85,B 0,C 180,E1 -29001.126,E2 -29001.126} C_VEL
LIN {X 0,Y 56.153,Z 426.414,A -85,B 0,C 180,E1 -29014.277,E2 -29014.277} C_VEL
LIN {X 0,Y 56.414,Z 419.914,A -85,B 0,C 180,E1 -29026.245,E2 -29026.245} C_VEL
LIN {X 0,Y 58.517,Z 412.216,A -85,B 0,C 180,E1 -29037.215,E2 -29037.215} C_VEL
LIN {X 0,Y 62.132,Z 402.753,A -85,B 0,C 180,E1 -29047.164,E2 -29047.164} C_VEL
LIN {X 0,Y 66.386,Z 392.618,A -85,B 0,C 180,E1 -29054.842,E2 -29054.842} C_VEL
LIN {X 0,Y 70.192,Z 383.565,A -85,B 0,C 180,E1 -29059.908,E2 -29059.908} C_VEL
LIN {X 0,Y 70.638,Z 382.077,A -85,B 0,C 180,E1 -29060.696,E2 -29060.696} C_VEL
LIN {X 0,Y 69.006,Z 373.218,A -85,B 0,C 180,E1 -29066.656,E2 -29066.656} C_VEL
LIN {X 0,Y 66.844,Z 364.757,A -85,B 0,C 180,E1 -29072.436,E2 -29072.436} C_VEL
LIN {X 0,Y 65.9,Z 361.181,A -85,B 0,C 180,E1 -29074.862,E2 -29074.862} C_VEL
LIN {X 0,Y 63.117,Z 355.576,A -85,B 0,C 180,E1 -29079.612,E2 -29079.612} C_VEL
LIN {X 0,Y 61.048,Z 351.637,A -85,B 0,C 180,E1 -29083.311,E2 -29083.311} C_VEL
LIN {X 0,Y 58.8,Z 348.733,A -85,B 0,C 180,E1 -29087.025,E2 -29087.025} C_VEL
LIN {X 0,Y 58.366,Z 347.215,A -85,B 0,C 180,E1 -29088.382,E2 -29088.382} C_VEL
LIN {X 0,Y 58.151,Z 347.236,A -85,B 0,C 180,E1 -29098.91,E2 -29098.91} C_VEL
LIN {X 0,Y 58.159,Z 347.236,A -85,B 0,C 180,E1 -29102.234,E2 -29102.234} C_VEL
LIN {X 0,Y 58.036,Z 347.249,A -85,B 0,C 180,E1 -29107.211,E2 -29107.211} C_VEL
LIN {X 0,Y 57.745,Z 347.299,A -85,B 0,C 180,E1 -29111.069,E2 -29111.069} C_VEL
LIN {X 0,Y 56.907,Z 347.408,A -85,B 0,C 180,E1 -29114.902,E2 -29114.902} C_VEL
LIN {X 0,Y 55.078,Z 347.632,A -85,B 0,C 180,E1 -29120.721,E2 -29120.721} C_VEL
LIN {X 0,Y 51.215,Z 348.103,A -85,B 0,C 180,E1 -29135.791,E2 -29135.791} C_VEL
LIN {X 0,Y 51.122,Z 348.1,A -85,B 0,C 180,E1 -29140.434,E2 -29140.434} C_VEL
LIN {X 0,Y 51.458,Z 348.074,A -85,B 0,C 180,E1 -29144.149,E2 -29144.149} C_VEL
LIN {X 0,Y 51.67,Z 348.047,A -85,B 0,C 180,E1 -29152.184,E2 -29152.184} C_VEL
LIN {X 0,Y 52.259,Z 347.972,A -85,B 0,C 180,E1 -29160.001,E2 -29160.001} C_VEL
LIN {X 0,Y 51.651,Z 348.047,A -85,B 0,C 180,E1 -29168.067,E2 -29168.067} C_VEL
LIN {X 0,Y 52.429,Z 350.652,A -85,B 0,C 180,E1 -29170.867,E2 -29170.867} C_VEL
LIN {X 0,Y 54.238,Z 353.1,A -85,B 0,C 180,E1 -29174.781,E2 -29174.781} C_VEL
LIN {X 0,Y 58.19,Z 360.954,A -85,B 0,C 180,E1 -29183.264,E2 -29183.264} C_VEL
LIN {X 0,Y 60.765,Z 367.077,A -85,B 0,C 180,E1 -29188.497,E2 -29188.497} C_VEL
LIN {X 0,Y 61.934,Z 373.255,A -85,B 0,C 180,E1 -29192.618,E2 -29192.618} C_VEL
LIN {X 0,Y 61.348,Z 379.053,A -85,B 0,C 180,E1 -29195.612,E2 -29195.612} C_VEL
LIN {X 0,Y 59.472,Z 390.739,A -85,B 0,C 180,E1 -29202.388,E2 -29202.388} C_VEL
LIN {X 0,Y 57.685,Z 401.405,A -85,B 0,C 180,E1 -29210.249,E2 -29210.249} C_VEL
LIN {X 0,Y 56.947,Z 405.858,A -85,B 0,C 180,E1 -29214.111,E2 -29214.111} C_VEL
LIN {X 0,Y 54.189,Z 412.805,A -85,B 0,C 180,E1 -29220.899,E2 -29220.899} C_VEL
LIN {X 0,Y 51.381,Z 421.344,A -85,B 0,C 180,E1 -29232.076,E2 -29232.076} C_VEL
LIN {X 0,Y 50.46,Z 428.195,A -85,B 0,C 180,E1 -29244.004,E2 -29244.004} C_VEL
LIN {X 0,Y 50.871,Z 432.692,A -85,B 0,C 180,E1 -29253.961,E2 -29253.961} C_VEL
LIN {X 0,Y 50.956,Z 436.504,A -85,B 0,C 180,E1 -29266.013,E2 -29266.013} C_VEL
LIN {X 0,Y 54.344,Z 440.238,A -85,B 0,C 180,E1 -29281.152,E2 -29281.152} C_VEL
LIN {X 0,Y 61.179,Z 442.646,A -85,B 0,C 180,E1 -29293.572,E2 -29293.572} C_VEL
LIN {X 0,Y 70.514,Z 443.859,A -85,B 0,C 180,E1 -29302.878,E2 -29302.878} C_VEL
LIN {X 0,Y 81.347,Z 443.849,A -85,B 0,C 180,E1 -29309.764,E2 -29309.764} C_VEL
LIN {X 0,Y 93.268,Z 442.624,A -85,B 0,C 180,E1 -29314.721,E2 -29314.721} C_VEL
LIN {X 0,Y 99.464,Z 441.545,A -85,B 0,C 180,E1 -29316.718,E2 -29316.718} C_VEL
LIN {X 0,Y 87.537,Z 442.278,A -85,B 0,C 180,E1 -29321.267,E2 -29321.267} C_VEL
LIN {X 0,Y 80.053,Z 442.013,A -85,B 0,C 180,E1 -29324.955,E2 -29324.955} C_VEL
LIN {X 0,Y 71.22,Z 440.906,A -85,B 0,C 180,E1 -29330.685,E2 -29330.685} C_VEL
LIN {X 0,Y 61.63,Z 438.241,A -85,B 0,C 180,E1 -29339.999,E2 -29339.999} C_VEL
LIN {X 0,Y 54.717,Z 434.518,A -85,B 0,C 180,E1 -29351.104,E2 -29351.104} C_VEL
LIN {X 0,Y 50.272,Z 429.371,A -85,B 0,C 180,E1 -29364.795,E2 -29364.795} C_VEL
LIN {X 0,Y 48.969,Z 422.823,A -85,B 0,C 180,E1 -29379.652,E2 -29379.652} C_VEL
LIN {X 0,Y 50.373,Z 415.212,A -85,B 0,C 180,E1 -29393.342,E2 -29393.342} C_VEL
LIN {X 0,Y 53.467,Z 406.708,A -85,B 0,C 180,E1 -29404.652,E2 -29404.652} C_VEL
LIN {X 0,Y 57.496,Z 397.664,A -85,B 0,C 180,E1 -29413.41,E2 -29413.41} C_VEL
LIN {X 0,Y 61.945,Z 387.767,A -85,B 0,C 180,E1 -29420.3,E2 -29420.3} C_VEL
LIN {X 0,Y 63.787,Z 383.606,A -85,B 0,C 180,E1 -29422.567,E2 -29422.567} C_VEL
LIN {X 0,Y 62.948,Z 376.96,A -85,B 0,C 180,E1 -29427.598,E2 -29427.598} C_VEL
LIN {X 0,Y 61.257,Z 369.059,A -85,B 0,C 180,E1 -29433.639,E2 -29433.639} C_VEL
LIN {X 0,Y 59.869,Z 363.916,A -85,B 0,C 180,E1 -29437.778,E2 -29437.778} C_VEL
LIN {X 0,Y 56.768,Z 357.705,A -85,B 0,C 180,E1 -29444.336,E2 -29444.336} C_VEL
LIN {X 0,Y 53.862,Z 352.846,A -85,B 0,C 180,E1 -29450.729,E2 -29450.729} C_VEL
LIN {X 0,Y 52.327,Z 351.421,A -85,B 0,C 180,E1 -29453.761,E2 -29453.761} C_VEL
LIN {X 0,Y 51.116,Z 348.616,A -85,B 0,C 180,E1 -29457.648,E2 -29457.648} C_VEL
LIN {X 0,Y 51.06,Z 348.121,A -85,B 0,C 180,E1 -29458.239,E2 -29458.239} C_VEL
LIN {X 0,Y 51.032,Z 348.129,A -85,B 0,C 180,E1 -29464.28,E2 -29464.28} C_VEL
LIN {X 0,Y 50.986,Z 348.125,A -85,B 0,C 180,E1 -29476.434,E2 -29476.434} C_VEL
LIN {X 0,Y 51.018,Z 348.124,A -85,B 0,C 180,E1 -29486.564,E2 -29486.564} C_VEL
LIN {X 0,Y 51.015,Z 348.128,A -85,B 0,C 180,E1 -29495.589,E2 -29495.589} C_VEL
LIN {X 0,Y 51.122,Z 348.1,A -85,B 0,C 180,E1 -29500.434,E2 -29500.434} C_VEL
LIN {X 0,Y 50.728,Z 348.368,A -85,B 0,C 180,E1 -29504.841,E2 -29504.841} C_VEL
LIN {X 0,Y 49.535,Z 349.091,A -85,B 0,C 180,E1 -29509.169,E2 -29509.169} C_VEL
LIN {X 0,Y 47.024,Z 352.02,A -85,B 0,C 180,E1 -29519.648,E2 -29519.648} C_VEL
LIN {X 0,Y 47.53,Z 353.647,A -85,B 0,C 180,E1 -29524.138,E2 -29524.138} C_VEL
LIN {X 0,Y 50.04,Z 358.453,A -85,B 0,C 180,E1 -29532.149,E2 -29532.149} C_VEL
LIN {X 0,Y 53.303,Z 365.784,A -85,B 0,C 180,E1 -29541.26,E2 -29541.26} C_VEL
LIN {X 0,Y 55.146,Z 370.846,A -85,B 0,C 180,E1 -29546.252,E2 -29546.252} C_VEL
LIN {X 0,Y 55.787,Z 376.233,A -85,B 0,C 180,E1 -29550.261,E2 -29550.261} C_VEL
LIN {X 0,Y 53.745,Z 387.068,A -85,B 0,C 180,E1 -29556.78,E2 -29556.78} C_VEL
LIN {X 0,Y 51.543,Z 397.988,A -85,B 0,C 180,E1 -29565.089,E2 -29565.089} C_VEL
LIN {X 0,Y 49.741,Z 406.395,A -85,B 0,C 180,E1 -29573.095,E2 -29573.095} C_VEL
LIN {X 0,Y 46.222,Z 414.613,A -85,B 0,C 180,E1 -29582.861,E2 -29582.861} C_VEL
LIN {X 0,Y 43.845,Z 422.622,A -85,B 0,C 180,E1 -29596.053,E2 -29596.053} C_VEL
LIN {X 0,Y 43.689,Z 429.016,A -85,B 0,C 180,E1 -29610,E2 -29610} C_VEL
LIN {X 0,Y 43.976,Z 430.803,A -85,B 0,C 180,E1 -29614.583,E2 -29614.583} C_VEL
LIN {X 0,Y 44.332,Z 434.835,A -85,B 0,C 180,E1 -29628.486,E2 -29628.486} C_VEL
LIN {X 0,Y 48.493,Z 438.847,A -85,B 0,C 180,E1 -29645.43,E2 -29645.43} C_VEL
LIN {X 0,Y 56.283,Z 441.521,A -85,B 0,C 180,E1 -29658.524,E2 -29658.524} C_VEL
LIN {X 0,Y 66.47,Z 442.979,A -85,B 0,C 180,E1 -29667.764,E2 -29667.764} C_VEL
LIN {X 0,Y 78.024,Z 443.25,A -85,B 0,C 180,E1 -29674.258,E2 -29674.258} C_VEL
LIN {X 0,Y 84.151,Z 442.944,A -85,B 0,C 180,E1 -29676.735,E2 -29676.735} C_VEL
LIN {X 0,Y 83.831,Z 442.89,A -85,B 0,C 180,E1 -29677.249,E2 -29677.249} C_VEL
LIN {X 0,Y 71.818,Z 441.968,A -85,B 0,C 180,E1 -29682.927,E2 -29682.927} C_VEL
LIN {X 0,Y 64.777,Z 440.684,A -85,B 0,C 180,E1 -29687.547,E2 -29687.547} C_VEL
LIN {X 0,Y 56.412,Z 438.197,A -85,B 0,C 180,E1 -29695.328,E2 -29695.328} C_VEL
LIN {X 0,Y 48.01,Z 433.688,A -85,B 0,C 180,E1 -29708.416,E2 -29708.416} C_VEL
LIN {X 0,Y 43.182,Z 428.134,A -85,B 0,C 180,E1 -29724.008,E2 -29724.008} C_VEL
LIN {X 0,Y 42.021,Z 420.86,A -85,B 0,C 180,E1 -29741.989,E2 -29741.989} C_VEL
LIN {X 0,Y 43.707,Z 413.47,A -85,B 0,C 180,E1 -29756.252,E2 -29756.252} C_VEL
LIN {X 0,Y 46.985,Z 405.433,A -85,B 0,C 180,E1 -29767.761,E2 -29767.761} C_VEL
LIN {X 0,Y 51.391,Z 396.29,A -85,B 0,C 180,E1 -29777.113,E2 -29777.113} C_VEL
LIN {X 0,Y 56.482,Z 385.794,A -85,B 0,C 180,E1 -29784.51,E2 -29784.51} C_VEL
LIN {X 0,Y 57.219,Z 384.068,A -85,B 0,C 180,E1 -29785.529,E2 -29785.529} C_VEL
LIN {X 0,Y 55.943,Z 375.233,A -85,B 0,C 180,E1 -29793.224,E2 -29793.224} C_VEL
LIN {X 0,Y 54.34,Z 367.726,A -85,B 0,C 180,E1 -29800.146,E2 -29800.146} C_VEL
LIN {X 0,Y 51.601,Z 361.742,A -85,B 0,C 180,E1 -29807.564,E2 -29807.564} C_VEL
LIN {X 0,Y 49.865,Z 358.656,A -85,B 0,C 180,E1 -29812.322,E2 -29812.322} C_VEL
LIN {X 0,Y 48.49,Z 357.126,A -85,B 0,C 180,E1 -29815.773,E2 -29815.773} C_VEL
LIN {X 0,Y 47.106,Z 354.035,A -85,B 0,C 180,E1 -29821.299,E2 -29821.299} C_VEL
LIN {X 0,Y 44.474,Z 351.182,A -85,B 0,C 180,E1 -29831.662,E2 -29831.662} C_VEL
LIN {X 0,Y 43.868,Z 349.012,A -85,B 0,C 180,E1 -29837.655,E2 -29837.655} C_VEL
LIN {X 0,Y 43.818,Z 349.02,A -85,B 0,C 180,E1 -29843.317,E2 -29843.317} C_VEL
LIN {X 0,Y 43.823,Z 349.02,A -85,B 0,C 180,E1 -29851.243,E2 -29851.243} C_VEL
LIN {X 0,Y 44.216,Z 348.97,A -85,B 0,C 180,E1 -29862.495,E2 -29862.495} C_VEL
LIN {X 0,Y 44.545,Z 349.126,A -85,B 0,C 180,E1 -29870.924,E2 -29870.924} C_VEL
LIN {X 0,Y 46.054,Z 351.769,A -85,B 0,C 180,E1 -29878.908,E2 -29878.908} C_VEL
LIN {X 0,Y 47.53,Z 353.647,A -85,B 0,C 180,E1 -29884.138,E2 -29884.138} C_VEL
LIN {X 0,Y 48.289,Z 355.52,A -85,B 0,C 180,E1 -29887.139,E2 -29887.139} C_VEL
LIN {X 0,Y 48.56,Z 359.21,A -85,B 0,C 180,E1 -29890.403,E2 -29890.403} C_VEL
LIN {X 0,Y 47.981,Z 367.605,A -85,B 0,C 180,E1 -29896.151,E2 -29896.151} C_VEL
LIN {X 0,Y 48.431,Z 370.737,A -85,B 0,C 180,E1 -29899.324,E2 -29899.324} C_VEL
LIN {X 0,Y 49.578,Z 375.014,A -85,B 0,C 180,E1 -29904.052,E2 -29904.052} C_VEL
LIN {X 0,Y 49.754,Z 377.753,A -85,B 0,C 180,E1 -29906.475,E2 -29906.475} C_VEL
LIN {X 0,Y 47.168,Z 388.727,A -85,B 0,C 180,E1 -29914.007,E2 -29914.007} C_VEL
LIN {X 0,Y 44.61,Z 399.116,A -85,B 0,C 180,E1 -29923.228,E2 -29923.228} C_VEL
LIN {X 0,Y 43.276,Z 404.797,A -85,B 0,C 180,E1 -29929.489,E2 -29929.489} C_VEL
LIN {X 0,Y 40.847,Z 410.075,A -85,B 0,C 180,E1 -29936,E2 -29936} C_VEL
LIN {X 0,Y 37.465,Z 418.836,A -85,B 0,C 180,E1 -29950.715,E2 -29950.715} C_VEL
LIN {X 0,Y 36.649,Z 425.897,A -85,B 0,C 180,E1 -29967.252,E2 -29967.252} C_VEL
LIN {X 0,Y 37.093,Z 428.798,A -85,B 0,C 180,E1 -29975.436,E2 -29975.436} C_VEL
LIN {X 0,Y 37.201,Z 430.421,A -85,B 0,C 180,E1 -29980.89,E2 -29980.89} C_VEL
LIN {X 0,Y 39.804,Z 435.357,A -85,B 0,C 180,E1 -30001.985,E2 -30001.985} C_VEL
LIN {X 0,Y 47.093,Z 438.972,A -85,B 0,C 180,E1 -30018.261,E2 -30018.261} C_VEL
LIN {X 0,Y 57.286,Z 441.319,A -85,B 0,C 180,E1 -30029.181,E2 -30029.181} C_VEL
LIN {X 0,Y 68.975,Z 442.469,A -85,B 0,C 180,E1 -30036.496,E2 -30036.496} C_VEL
LIN {X 0,Y 68.266,Z 442.241,A -85,B 0,C 180,E1 -30037.906,E2 -30037.906} C_VEL
LIN {X 0,Y 56.233,Z 439.575,A -85,B 0,C 180,E1 -30045.524,E2 -30045.524} C_VEL
LIN {X 0,Y 46.696,Z 435.915,A -85,B 0,C 180,E1 -30055.683,E2 -30055.683} C_VEL
LIN {X 0,Y 39.232,Z 430.906,A -85,B 0,C 180,E1 -30070.318,E2 -30070.318} C_VEL
LIN {X 0,Y 35.276,Z 424.446,A -85,B 0,C 180,E1 -30089.508,E2 -30089.508} C_VEL
LIN {X 0,Y 35.347,Z 417.346,A -85,B 0,C 180,E1 -30108.21,E2 -30108.21} C_VEL
LIN {X 0,Y 37.802,Z 410.214,A -85,B 0,C 180,E1 -30122.609,E2 -30122.609} C_VEL
LIN {X 0,Y 42.196,Z 401.235,A -85,B 0,C 180,E1 -30135.321,E2 -30135.321} C_VEL
LIN {X 0,Y 47.511,Z 391.077,A -85,B 0,C 180,E1 -30144.779,E2 -30144.779} C_VEL
LIN {X 0,Y 50.485,Z 385.368,A -85,B 0,C 180,E1 -30148.584,E2 -30148.584} C_VEL
LIN {X 0,Y 50.24,Z 380.866,A -85,B 0,C 180,E1 -30153.01,E2 -30153.01} C_VEL
LIN {X 0,Y 49.186,Z 372.99,A -85,B 0,C 180,E1 -30161.223,E2 -30161.223} C_VEL
LIN {X 0,Y 48.281,Z 370.049,A -85,B 0,C 180,E1 -30164.884,E2 -30164.884} C_VEL
LIN {X 0,Y 46.644,Z 366.254,A -85,B 0,C 180,E1 -30170.612,E2 -30170.612} C_VEL
LIN {X 0,Y 45.131,Z 363.522,A -85,B 0,C 180,E1 -30175.946,E2 -30175.946} C_VEL
LIN {X 0,Y 43.784,Z 360.786,A -85,B 0,C 180,E1 -30181.986,E2 -30181.986} C_VEL
LIN {X 0,Y 43.08,Z 359.593,A -85,B 0,C 180,E1 -30185.347,E2 -30185.347} C_VEL
LIN {X 0,Y 41.679,Z 357.853,A -85,B 0,C 180,E1 -30192.415,E2 -30192.415} C_VEL
LIN {X 0,Y 41.311,Z 356.313,A -85,B 0,C 180,E1 -30197.119,E2 -30197.119} C_VEL
LIN {X 0,Y 40.412,Z 355.263,A -85,B 0,C 180,E1 -30210.407,E2 -30210.407} C_VEL
LIN {X 0,Y 40.656,Z 355.262,A -85,B 0,C 180,E1 -30219.775,E2 -30219.775} C_VEL
LIN {X 0,Y 41.985,Z 356.125,A -85,B 0,C 180,E1 -30230.365,E2 -30230.365} C_VEL
LIN {X 0,Y 43.972,Z 359.544,A -85,B 0,C 180,E1 -30241.489,E2 -30241.489} C_VEL
LIN {X 0,Y 45.641,Z 363.374,A -85,B 0,C 180,E1 -30248.859,E2 -30248.859} C_VEL
LIN {X 0,Y 47.829,Z 369.026,A -85,B 0,C 180,E1 -30257.092,E2 -30257.092} C_VEL
LIN {X 0,Y 48.431,Z 370.737,A -85,B 0,C 180,E1 -30259.324,E2 -30259.324} C_VEL
LIN {X 0,Y 48.595,Z 373.283,A -85,B 0,C 180,E1 -30261.604,E2 -30261.604} C_VEL
LIN {X 0,Y 47.832,Z 376.179,A -85,B 0,C 180,E1 -30263.193,E2 -30263.193} C_VEL
LIN {X 0,Y 46.187,Z 379.646,A -85,B 0,C 180,E1 -30264.55,E2 -30264.55} C_VEL
LIN {X 0,Y 42.037,Z 386.814,A -85,B 0,C 180,E1 -30267.553,E2 -30267.553} C_VEL
LIN {X 0,Y 41.079,Z 389.154,A -85,B 0,C 180,E1 -30269.323,E2 -30269.323} C_VEL
LIN {X 0,Y 37.892,Z 399.634,A -85,B 0,C 180,E1 -30280.086,E2 -30280.086} C_VEL
LIN {X 0,Y 36.214,Z 405.142,A -85,B 0,C 180,E1 -30287.216,E2 -30287.216} C_VEL
LIN {X 0,Y 32.06,Z 413.349,A -85,B 0,C 180,E1 -30300.447,E2 -30300.447} C_VEL
LIN {X 0,Y 29.757,Z 421.363,A -85,B 0,C 180,E1 -30319.797,E2 -30319.797} C_VEL
LIN {X 0,Y 30.247,Z 426.677,A -85,B 0,C 180,E1 -30336.672,E2 -30336.672} C_VEL
LIN {X 0,Y 30.553,Z 428.362,A -85,B 0,C 180,E1 -30343.299,E2 -30343.299} C_VEL
LIN {X 0,Y 34.137,Z 433.641,A -85,B 0,C 180,E1 -30368.143,E2 -30368.143} C_VEL
LIN {X 0,Y 42.762,Z 437.535,A -85,B 0,C 180,E1 -30385.262,E2 -30385.262} C_VEL
LIN {X 0,Y 54.014,Z 440.16,A -85,B 0,C 180,E1 -30395.617,E2 -30395.617} C_VEL
LIN {X 0,Y 55.076,Z 440.219,A -85,B 0,C 180,E1 -30397.491,E2 -30397.491} C_VEL
LIN {X 0,Y 43.212,Z 436.114,A -85,B 0,C 180,E1 -30407.381,E2 -30407.381} C_VEL
LIN {X 0,Y 35.092,Z 431.597,A -85,B 0,C 180,E1 -30419.998,E2 -30419.998} C_VEL
LIN {X 0,Y 29.599,Z 426.026,A -85,B 0,C 180,E1 -30438.239,E2 -30438.239} C_VEL
LIN {X 0,Y 28.015,Z 418.189,A -85,B 0,C 180,E1 -30463.957,E2 -30463.957} C_VEL
LIN {X 0,Y 30.921,Z 409.634,A -85,B 0,C 180,E1 -30485.385,E2 -30485.385} C_VEL
LIN {X 0,Y 36.405,Z 399.594,A -85,B 0,C 180,E1 -30501.056,E2 -30501.056} C_VEL
LIN {X 0,Y 42.905,Z 388.393,A -85,B 0,C 180,E1 -30511.456,E2 -30511.456} C_VEL
LIN {X 0,Y 44.235,Z 385.874,A -85,B 0,C 180,E1 -30513.162,E2 -30513.162} C_VEL
LIN {X 0,Y 43.822,Z 379.144,A -85,B 0,C 180,E1 -30521.192,E2 -30521.192} C_VEL
LIN {X 0,Y 43.573,Z 376.34,A -85,B 0,C 180,E1 -30524.596,E2 -30524.596} C_VEL
LIN {X 0,Y 42.511,Z 372.714,A -85,B 0,C 180,E1 -30530.376,E2 -30530.376} C_VEL
LIN {X 0,Y 41.427,Z 369.89,A -85,B 0,C 180,E1 -30535.997,E2 -30535.997} C_VEL
LIN {X 0,Y 39.796,Z 366.16,A -85,B 0,C 180,E1 -30545.488,E2 -30545.488} C_VEL
LIN {X 0,Y 38.34,Z 363.286,A -85,B 0,C 180,E1 -30557.158,E2 -30557.158} C_VEL
LIN {X 0,Y 37.882,Z 362.117,A -85,B 0,C 180,E1 -30566.182,E2 -30566.182} C_VEL
LIN {X 0,Y 37.98,Z 361.865,A -85,B 0,C 180,E1 -30578.28,E2 -30578.28} C_VEL
LIN {X 0,Y 39.107,Z 362.801,A -85,B 0,C 180,E1 -30589.648,E2 -30589.648} C_VEL
LIN {X 0,Y 40.456,Z 365.914,A -85,B 0,C 180,E1 -30600.001,E2 -30600.001} C_VEL
LIN {X 0,Y 41.534,Z 369.489,A -85,B 0,C 180,E1 -30607.292,E2 -30607.292} C_VEL
LIN {X 0,Y 42.846,Z 373.569,A -85,B 0,C 180,E1 -30614.245,E2 -30614.245} C_VEL
LIN {X 0,Y 43.912,Z 377.843,A -85,B 0,C 180,E1 -30620.158,E2 -30620.158} C_VEL
LIN {X 0,Y 43.949,Z 379.294,A -85,B 0,C 180,E1 -30621.642,E2 -30621.642} C_VEL
LIN {X 0,Y 41.079,Z 389.154,A -85,B 0,C 180,E1 -30629.323,E2 -30629.323} C_VEL
LIN {X 0,Y 38.994,Z 393.987,A -85,B 0,C 180,E1 -30633.329,E2 -30633.329} C_VEL
LIN {X 0,Y 35.992,Z 398.551,A -85,B 0,C 180,E1 -30637.107,E2 -30637.107} C_VEL
LIN {X 0,Y 28.974,Z 406.869,A -85,B 0,C 180,E1 -30646.633,E2 -30646.633} C_VEL
LIN {X 0,Y 25.277,Z 412.112,A -85,B 0,C 180,E1 -30657.084,E2 -30657.084} C_VEL
LIN {X 0,Y 22.838,Z 419.984,A -85,B 0,C 180,E1 -30681.149,E2 -30681.149} C_VEL
LIN {X 0,Y 23.444,Z 424.426,A -85,B 0,C 180,E1 -30698.621,E2 -30698.621} C_VEL
LIN {X 0,Y 24.003,Z 426.26,A -85,B 0,C 180,E1 -30707.026,E2 -30707.026} C_VEL
LIN {X 0,Y 26.25,Z 429.846,A -85,B 0,C 180,E1 -30726.559,E2 -30726.559} C_VEL
LIN {X 0,Y 33.759,Z 434.057,A -85,B 0,C 180,E1 -30746.38,E2 -30746.38} C_VEL
LIN {X 0,Y 39.214,Z 435.963,A -85,B 0,C 180,E1 -30753.652,E2 -30753.652} C_VEL
LIN {X 0,Y 41.155,Z 436.409,A -85,B 0,C 180,E1 -30757.529,E2 -30757.529} C_VEL
LIN {X 0,Y 30.216,Z 430.97,A -85,B 0,C 180,E1 -30770.974,E2 -30770.974} C_VEL
LIN {X 0,Y 23.021,Z 424.696,A -85,B 0,C 180,E1 -30792.989,E2 -30792.989} C_VEL
LIN {X 0,Y 20.945,Z 417.66,A -85,B 0,C 180,E1 -30822.147,E2 -30822.147} C_VEL
LIN {X 0,Y 23.227,Z 410.758,A -85,B 0,C 180,E1 -30845.187,E2 -30845.187} C_VEL
LIN {X 0,Y 28.317,Z 402.13,A -85,B 0,C 180,E1 -30863.08,E2 -30863.08} C_VEL
LIN {X 0,Y 34.259,Z 392.965,A -85,B 0,C 180,E1 -30873.908,E2 -30873.908} C_VEL
LIN {X 0,Y 38.079,Z 386.631,A -85,B 0,C 180,E1 -30878.852,E2 -30878.852} C_VEL
